REGION Network 2: Block description — Sections 3.2 to 3.7
   // ▂▂▂▂▂▂▂▂▂▂▂▂▂▂▂▂▂▂▂▂▂▂▂▂▂▂▂▂▂▂▂▂▂▂▂▂▂▂▂▂▂▂▂▂
   // 3.2     Warnings and alarms
   // 
   // By default, the block generates 4 alarms and warnings (2 warnings and 2 alarms, 4 in total) 
   // as follows:
   // 
   // 
   //  ――――――――――――――――――――――――――――――――――――――――――
   //  ALARM / WARNING     FUNCTION
   //  ――――――――――――――――――――――――――――――――――――――――――
   //  Alarm high       Scaled signal is equal to or above a preset alarm high setpoint
   //  Warning high      Scaled signal is equal to or above a preset warning high setpoint
   //  Warning low     Scaled signal is equal to or below a preset warning low setpoint
   //  Alarm low      Scaled signal is equal to or below a preset alarm low setpoint
   //  ――――――――――――――――――――――――――――――――――――――――――
   //  Default alarm and warning signals
   // 
   // 
   // The active state of any alarm or warning is stored in the DATA_DYNAMIC structure in the following 
   // variables:
   // 
   //  UT22001_Dy_InstAnalogRead
   //  ――――――――――――――――――――――――――――――――――――――――――
   //  SIGNAL NAME          FUNCTION                     TYPE
   //  ――――――――――――――――――――――――――――――――――――――――――
   //  msg_Alm_H         MESSAGE — Alarm - high alarm is active        Bool
   //  msg_Alm_L          MESSAGE — Alarm - low alarm is active          Bool
   //  msg_Wrn_H          MESSAGE — Warning - high warning is active      Bool
   //  msg_Wrn_L          MESSAGE — Warning - low warning is active        Bool
   //  ――――――――――――――――――――――――――――――――――――――――――
   // 
   // The alarms and warnings that end with _H are activated when the scaled instrument reading is 
   // greater than or equal to a setpoint threshold (i.e. activate when the measured quantity is too 
   // high; generally, if there is both an alarm high and a warning high, the convention within the PAL 
   // is that the warning should activate before the alarm².
   // 
   // 
   // The alarms and warnings that end with _L are activated when the scaled instrument reading is 
   // less than or equal to a setpoint threshold (i.e. activate when the measured quantity is too high; 
   // generally, if there is both an alarm low and a warning low, the convention within the PAL is that 
   // the warning should activate before the alarm².
   // 
   // ――――――――――
   // ²         This is just a convention, there is nothing to stop the warning being set to occur after 
   //      the alarm (i.e. the warning detecting the most extreme condition). All alarms and 
   //      warnings are entirely independent of each other and no error checking is carried 
   //      out to ensure that any particular threshold is above or below another.
   // ――――――――――
   // 
   // All alarms and warnings are individually enabled (a disabled alarm or warning will never be 
   // activated), all alarms and warnings have individual setpoint values (the value at which the 
   // alarm or warning is triggered), all alarms and warnings have individual hysteresis valves 
   // (effectively a tolerance band, the difference between where an alarm activates and where is 
   // deactivates, used to prevent nuisance or “chattering” alarms). Finally, each alarm and warning 
   // has a configurable on and off delay (the alarm or warning will only activate if the reading is 
   // outside the threshold for the on-delay time and similarly will only deactivate when the reading 
   // is inside the threshold and hysteresis for the off-delay time).
   // 
   // The following table summarises all the available signals for each alarm and warning:
   // 
   //  ――――――――――――――――――――――――――――――――――――――――――
   //  SIGNAL          FUNCTION             TYPE   DETAILS
   //  ――――――――――――――――――――――――――――――――――――――――――
   //  CONFIG_XXX_Y_ENABLE Alarm/warning enabled      Bool    1 = enabled, 0 = disabled
   //  SP_XXX_Y_VAL      Alarm/warning setpoint value    Real Engineering units
   //  SP_XXX_Y_HYST_VAL    Alarm/warning hysteresis value Real Engineering units
   //  TIME_XXX_Y_ON_DEL   Alarm/warning on delay time   Real In seconds
   //  TIME_XXX_Y_OFF_DEL     Alarm/warning off delay time   Real In seconds
   //  mode_Xxx_Y_MaskOn     Alarm/warning is masked      Bool    1 = masked, 0 = normal
   //  msg_Xxx_Y         Alarm/warning is active      Bool    1 = active, 0 = inactive
   //  ――――――――――――――――――――――――――――――――――――――――――
   //  Default alarm and warning signals — where XXX is either ALM or WRN and Y is either H or L
   // 
   // 
   // 
   // ▁▁▁▁▁▁▁▁▁▁▁▁▁▁▁▁▁▁▁▁▁▁▁▁▁▁▁▁▁▁▁▁▁▁▁▁▁▁▁▁▁▁▁▁
   // 3.2.1     High alarms and warnings (an example)
   // 
   // This example explains how a high alarm signal is generated, a high warning works in exactly the 
   // same way with WRN being substituted for ALM.
   // 
   // The full set of signals associated with the high alarm are:
   // 
   //  ――――――――――――――――――――――――――――――――――――――――――
   //  SIGNAL           FUNCTION            TYPE   DETAILS
   //  ――――――――――――――――――――――――――――――――――――――――――
   //  SP_ALM_H_VAL      Alarm high setpoint value    Real Engineering units
   //  SP_ALM_H_HYST_VAL    Alarm high hysteresis value Real Engineering units
   //  TIME_ALM_H_ON_DEL   Alarm high on delay time   Real In seconds
   //  TIME_ALM_H_OFF_DEL     Alarm high off delay time   Real In seconds
   //  mode_Alm_H_MaskOn    Alarm is masked         Bool    1 = masked, 0 = normal
   //  msg_Alm_H        Alarm high is active      Bool    1 = active, 0 = inactive
   //  ――――――――――――――――――――――――――――――――――――――――――
   // 
   // The figure below indicates how each of these signal functions (note TIME_ALM_H_ON_DEL and
   // TIME_ALM_H_OFF_DEL have been abbreviated to ON_DEL and OFF_DEL respectively):
   // 
   // 
   //                 │
   //                 │          ╱╲╱╲
   //                 │    ①      ②╱    ╲
   //       SP_ALM_H_VAL↘│____╱╲________╱____________╲③_______④__________ 
   //    SP_ALM_H_HYST_VAL ↕│__╱____╲____╱╎_____╎_______╲____╱╲___________
   //                 │╱    ╲╱ ╎    ╎      ╲╱     ╲
   //                 │        ╎    ╎          ╎╲
   //                 │        ╎    ╎          ╎ ╲___
   //                 │        ╎    ╎          ╎    ╎╲╱
   //                 │    ON_DEL→╎    ╎←    OFF_DEL→╎    ╎←
   //                 ┼─────────────────────────────
   // 
   //                            ╎                        ╎
   // 
   //         msg_Alm_H │             ┏━━━━━━━━━━━━┓
   //                 │             ┃               ┃
   // CONFIG_ALM_H_ENABLE = 1  │             ┃   ALARM IS ACTIVE    ┃
   // & mode_Alm_H_MaskOn = 0 │             ┃               ┃
   //                 │             ┃               ┃
   //                 ┼━━━━━━━━━━━━╶╶╶╶╶╶╶╶╶╶╶╶╶━━━━
   // 
   //                            ╎                        ╎
   // 
   //         msg_Alm_H │          
   // ⑤               │             ╎               ╎             
   // CONFIG_ALM_H_ENABLE = 0  │             
   //     OR          │             ╎               ╎
   // CONFIG_ALM_H_ENABLE = 1  │          
   // & mode_Alm_H_MaskOn = 1 ┼━━━━━━━━━━━━━━━━━━━━━━━━━━━━━
   // 
   // 
   // 
   // ▁▁▁▁▁▁▁▁▁▁▁▁▁▁▁▁▁▁▁▁▁▁▁▁▁▁▁▁▁▁▁▁▁▁▁▁▁▁▁▁▁▁▁▁
   // Scenario ①, alarm setpoint reached, but for less than on-delay duration
   // 
   // The graph represents the scaled analogue instrument reading, actual_Value (in engineering 
   // units). The top horizontal line is the setpoint for the high alarm (SP_ALM_H_VAL).
   // 
   // If the alarm is enabled (CONFIG_ALM_H_ENABLE = 1) then the following actions occur:
   // 
   // At point ① on the graph, the signal actual_Value reaches (and exceeds) the threshold value 
   // SP_ALM_H_VAL; i.e.:
   // 
   //           actual_Value ≥ SP_ALM_H_VAL
   // 
   // At this point, the alarm setpoint is exceeded and the on-delay timer starts; in the case of point ①, 
   // the signal actual_Value falls back below the setpoint value before the on-delay timer reaches 
   // the time set in TIME_ALM_H_ON_DEL, consequently the alarm does not activate.
   // 
   // 
   // 
   // ▁▁▁▁▁▁▁▁▁▁▁▁▁▁▁▁▁▁▁▁▁▁▁▁▁▁▁▁▁▁▁▁▁▁▁▁▁▁▁▁▁▁▁▁
   // Scenario ②, alarm setpoint reached for more than the on-delay duration
   // 
   // At point ② on the graph, the signal actual_Value again reaches (and exceeds) the setpoint value 
   // SP_ALM_H_VAL.
   // 
   // Again, at this point, the alarm threshold is exceeded and the on-delay timer starts; in the case of 
   // point ②, the signal actual_Value remains at or above the setpoint value for the full duration of 
   // the TIME_ALM_H_ON_DEL and consequently the alarm activates (msg_Alm_H goes to a high 
   // state), this is indicated in the middle msg_Alm_H graph.
   // 
   // 
   // 
   // ▁▁▁▁▁▁▁▁▁▁▁▁▁▁▁▁▁▁▁▁▁▁▁▁▁▁▁▁▁▁▁▁▁▁▁▁▁▁▁▁▁▁▁▁
   // Scenario ③, alarm reset level reached, but for less than the off-delay duration
   // 
   // At point ③, the signal actual_Value falls to the point at which the alarm is no longer active i.e.:
   // 
   //           actual_Value < (SP_ALM_H_VAL − SP_ALM_H_HYST_VAL)
   // 
   // Note:    in this case the inequality is less than (not less than or equal to), this is to prevent 
   //      conflict detecting the threshold and detecting the reset value if SP_ALM_H_HYST_VAL 
   //      is set to zero.
   // 
   // At this point, the signal is below the alarm reset level:
   // 
   //           SP_ALM_H_VAL − SP_ALM_H_HYST_VAL
   // 
   // and the off-delay timer starts; in the case of point 3, the signal actual_Value re-turns above the 
   // reset threshold before the off-delay timer reaches the time set in TIME_ALM_H_OFF_DEL, 
   // consequently, the alarm does not deactivate.
   // 
   // 
   // 
   // ▁▁▁▁▁▁▁▁▁▁▁▁▁▁▁▁▁▁▁▁▁▁▁▁▁▁▁▁▁▁▁▁▁▁▁▁▁▁▁▁▁▁▁▁
   // Scenario ④, alarm reset level reached for more than the off-delay duration
   // 
   // At point ④ on the graph, the signal actual_Value again falls below the alarm reset level 
   // (SP_ALM_H_VAL − SP_ALM_H_HYST_VAL).
   // 
   // Again, at this point, the off-delay timer starts; in the case of point ④, the signal actual_Value 
   // remains below the reset threshold for the full duration of the TIME_ALM_H_OFF_DEL and 
   // consequently, the alarm deactivates (msg_Alm_H goes to a low state), this is indicated in the 
   // middle msg_Alm_H graph.
   // 
   // 
   // 
   // ▁▁▁▁▁▁▁▁▁▁▁▁▁▁▁▁▁▁▁▁▁▁▁▁▁▁▁▁▁▁▁▁▁▁▁▁▁▁▁▁▁▁▁▁
   // Scenario ⑤, alarm is disabled
   // 
   // If the alarm is disabled (CONFIG_ALM_H_ENABLE = 0) then the alarm will never activate 
   // (msg_Alm_H is always in a low state), this is indicated in the lower msg_Alm_H graph.
   // 
   // Note:    The timer for disabled alarms and warnings is permanently set to zero.
   // 
   // 
   // ▁▁▁▁▁▁▁▁▁▁▁▁▁▁▁▁▁▁▁▁▁▁▁▁▁▁▁▁▁▁▁▁▁▁▁▁▁▁▁▁▁▁▁▁
   // 3.2.2     Low alarms and warnings
   // 
   // Low alarms and warnings are very similar to the high alarms of § 3.2.1, they do however work
   // in the opposite sense (the inequalities are reversed), low alarms and warnings are activated
   // when the actual_Value falls below, or is equal to, the SP_ALM_L_VAL, and deactivates when it
   // rises above SP_ALM_L_VAL + SP_ALM_L_HYST_VAL.
   // 
   // On and off delays work in exactly the same way as those for the high alarm.
   // 
   // A worked example of the low alarm is given in the online documentation for this block:
   // 
   // select this block in the project tree and press:
   //      SHIFT + F1
   // 
   // 
   // 
   // 
   // ▁▁▁▁▁▁▁▁▁▁▁▁▁▁▁▁▁▁▁▁▁▁▁▁▁▁▁▁▁▁▁▁▁▁▁▁▁▁▁▁▁▁▁▁
   // 3.2.3     Masking alarms and warnings
   // 
   // There are conditions where it can become necessary to mask (supress) alarms and warnings, a 
   // typical example could be a flow meter that monitors the flow into a filter; under normal 
   // conditions the flow meter would generate a low alarm if the flow into the filter were below a 
   // certain setpoint (indicating that the filter is becoming blocked).
   // 
   // It would be normal practice to supress this alarm when the filter was being cleaned, under 
   // these circumstances there would be no flow into the filter, but this would be a normal operating 
   // condition for the filter; the flow meter should only be monitoring for a low alarm during normal 
   // operation, not when the filter is being cleaned.
   // 
   // This suppression of an alarm or warning is referred to as “masking”, and there is a mask bit for 
   // each alarm and warning:
   // 
   //  ――――――――――――――――――――――――――――――――――――――――――
   //  SIGNAL           FUNCTION           TYPE   DETAILS
   //  ――――――――――――――――――――――――――――――――――――――――――
   //  mode_Alm_H_MaskOn    Masks the high alarm     Bool    1 = alarm masked, 0 = normal
   //  mode_Alm_L_MaskOn    Masks the low alarm    Bool    1 = alarm masked, 0 = normal
   //  mode_Wrn_H_MaskOn    Masks the high warning    Bool    1 = warning masked, 0 = normal
   //  mode_Wrn_L_MaskOn     Masks the low warning      Bool    1 = warning masked, 0 = normal
   //  ――――――――――――――――――――――――――――――――――――――――――
   //  Alarm and warning mask signals
   // 
   //  
   // Any alarm or warning that is masked (the mode_Xxx_Y_MaskOn = 1), will deactivate instantly 
   // (there is no off-delay) and will not reactivate activate (the msg_Xxx_Y will be set to zero), the 
   // effect is the same as if the CONFIG_XXX_Y_ENABLE bit were turned off.
   // 
   // The difference between the mask and the ENABLE signals is that the enable signal is a 
   // configuration of the instrument (it determines which alarms and warnings are configured for the 
   // particular instrument) and does not change at run-time (it is stored in static data block).
   // 
   // The mask signal on the other hand can be changed at run-time (either by some aspect of the 
   // Controller program or by the operator). The mask signal is stored in a dynamic data block and 
   // can be freely modified.
   // 
   // Note:    If an alarm or warning is not enabled (CONFIG_XXX_Y_ENABLE = 0), then the mask bit 
   //      (mode_Xxx_Y_MaskOn) will not do anything (setting it will not enable the alarm), in 
   //      fact if the alarm or warning is not enabled, the mask bit will be permanently set to 
   //      zero.
   // 
   // Masking alarms and warnings is the correct way to disable an alarm as part of the process 
   // operation of the plant.
   // 
   // When an alarm or warning goes from a masked condition to an unmasked condition (returns to 
   // normal operation), the on-delay timer will be reset and any alarm or warning condition will 
   // have to go back through the on-delay process before the alarm or warning can reactivate, this is 
   // true even if the alarm were active before being masked.
   // 
   // 
   // 
   // 
   // ▁▁▁▁▁▁▁▁▁▁▁▁▁▁▁▁▁▁▁▁▁▁▁▁▁▁▁▁▁▁▁▁▁▁▁▁▁▁▁▁▁▁▁▁
   // 3.2.4     A note on dynamically enabling alarms
   // 
   // In normal operations, alarms are either enabled or disabled as part of the instrument 
   // configuration and this configuration will not change during run-time; the enable signal 
   // (CONFIG_XXX_Y_ENABLE) is after all in a static data block. 
   // 
   // However, it is possible that the static data block is being used as a recipe block and as such it 
   // could be overloaded at some point during run-time.
   // 
   // Should the block detect a change in any of the CONFIG_XXX_Y_ENABLE; specifically, a rising 
   // edge, the block provided error checking to ensure that the associated alarm/warning timer 
   // (actual_Xxx_Y_Timer) is preset to correct TIME_XXX_Y_ON_DEL, this prevents the alarm/warning 
   // from activating instantly, if the actual_Value is outside the alarm/warning setpoint. A condition 
   // that could arise because the timer is set to zero while ever the alarm/warning is disabled.
   // 
   // Note:    This is a minor technical point, but it is a necessary error trapping mechanism — the 
   //      situation could arise even if it is unlikely.
   // 
   // 
   // 
   // ▂▂▂▂▂▂▂▂▂▂▂▂▂▂▂▂▂▂▂▂▂▂▂▂▂▂▂▂▂▂▂▂▂▂▂▂▂▂▂▂▂▂▂▂
   // 3.3     Fault signals
   // 
   // There are four fault signals that can be produced by the block:
   // 
   // 
   //  ――――――――――――――――――――――――――――――――――――――――――
   //  SIGNAL           FUNCTION            TYPE   DETAILS
   //  ――――――――――――――――――――――――――――――――――――――――――
   //  msg_Flt_UnderRange   The instrument is more than   Bool    1 = under range, 0 = healthy
   //                 a percentage below the its 
   //                 minimum value
   //  msg_Flt_OverRange     The instrument is more than   Bool    1 = over range, 0 = healthy
   //                 a percentage above its 
   //                 maximum value
   //  msg_Flt_OutOfRange   Common fault, either       Bool    1 = out of range, 0 = healthy
   //                 under or over range
   //  msg_Flt_External     The instrument itself is    Bool    1 = fault, 0 = healthy
   //                 indicating a fault 
   //                 (hardwired signal)
   //  ――――――――――――――――――――――――――――――――――――――――――
   //  Block fault signals 
   // 
   // 
   // 
   // ▁▁▁▁▁▁▁▁▁▁▁▁▁▁▁▁▁▁▁▁▁▁▁▁▁▁▁▁▁▁▁▁▁▁▁▁▁▁▁▁▁▁▁▁
   // 3.3.1     Over, under and out of range fault signals
   // 
   // If the signal from the instrument the RAW_ANALOG signal, is outside the RANGE_RAW_MIN to 
   // RANGE_RAW_MAX range (red dotted area of the graph, Figure 3.1), the scaled instrument reading 
   // (actual_Value) will still be calculated correctly; however, an appropriate, over-range or 
   // under-range (msg_Flt_OverRange or msg_Flt_UnderRange) signal will be generated to indicate 
   // that the instrument signal is outside of its calibrated range and is potentially no longer accurate.
   // 
   // Some tolerance is permitted before either the msg_Flt_OverRange or msg_Flt_UnderRange 
   // signals is activated (this is to prevent nuisance alarms — most instruments are tolerant of slight 
   // over and under shoot readings). 
   // 
   // The tolerance applied to the out of range signals is a percentage of the raw range of the 
   // instrument (the raw range being RANGE_RAW_MAX − RANGE_RAW_MIN). 
   // 
   // The tolerance to be applied is given in the parameter RANGE_OOR_PERCENT, this is a real 
   // (floating point) number in the range 0.0-10.0%.
   // 
   // If the tolerance for the instrument is not known, a generic value of 2.5% should be used.
   // 
   // The out of range tolerance absolute value (in terms of the RAW_ANALOG rather than as a 
   // percentage) is calculated as:
   // 
   // 
   // 
   // ┌─────────────────────────────────────┐
   // │                            (RANGE_RAW_MAX ─ RANGE_RAW_MIN) ╳ RANGE_OOR_PERCENT  │
   // │ calcRawOOR =  ―――――――――――――――――――――――――――― │
   // │                      100              │
   // └─────────────────────────────────────┘
   // 
   // Thus, if RANGE_RAW_MIN is 0, RANGE_RAW_MAX is 27648 and a RANGE_OOR_PERCENT of 2.5% is 
   // selected, the absolute out of range value (calcRawOOR in the above equation) has a calculated
   //  value of 691. 
   // 
   // In this example, the msg_Flt_OverRange signal would activate when RAW_ANALOG 
   // exceeded a value of RANGE_RAW_MAX + 691 (or 28,339). The msg_Flt_UnderRange signal would 
   // activate when RAW_ANALOG fell below a value of RANGE_RAW_MIN − 691 (or −691).
   // 
   // The RANGE_OOR_PERCENT is applied directly to the RAW_ANALOG signal, however, because the 
   // instrument is considered to be linear, the same calculation can also be ap-plied directly to the 
   // scaled reading of the instrument (actual_Value). 
   // 
   // In the example given in § 2.1, the instrument spans the range of -100 l/s to +100 l/s 
   // (i.e. RANGE_SCALE_MIN = -100 and RANGE_SCALE_MAX = +100) then the scaled range of the 
   // instrument is 200 l/s (RANGE_SCALE_MAX − RANGE_SCALE_MIN) and the absolute out of range 
   // value would be 2.5% of the scaled range (or 5 l/s). thus, the msg_Flt_OverRange signal would 
   // activate above 105 l/s and the msg_Flt_UnderRange signal would activate below −105 l/s.
   // 
   // Note:    If the range information supplied to the module is incorrect, either:
   //        •   RAW_MAX <= RAW_MIN or
   //        •   SCALE_MAX <= SCALE_MIN
   //      Then all the out of range signals are activated
   // 
   // 
   // 
   // ▁▁▁▁▁▁▁▁▁▁▁▁▁▁▁▁▁▁▁▁▁▁▁▁▁▁▁▁▁▁▁▁▁▁▁▁▁▁▁▁▁▁▁▁
   // Common out of range signal
   // 
   // There is a third out of range signal: msg_Flt_OutOfRange, this signal is a common signal that 
   // just indicates the instrument is out of its calibrated range (it does not specify whether it is over 
   // or under range). It is activated if either the msg_Flt_OverRange or msg_Flt_UnderRange signal is 
   // active.
   // 
   // 
   // 
   // ▁▁▁▁▁▁▁▁▁▁▁▁▁▁▁▁▁▁▁▁▁▁▁▁▁▁▁▁▁▁▁▁▁▁▁▁▁▁▁▁▁▁▁▁
   // 3.3.2     External fault signal
   // 
   // The external fault is an optional hardwired signal from the instrument, it indicates that the 
   // instrument itself is registering that there is some problem. Such external fault signals are more 
   // commonly associated with complex instruments (mass flow metres, ultrasonic level 
   // transducers, analytical instruments &c.) rather than the more simplistic instruments (pressure 
   // sensors, temperature transmitters &c.).
   // 
   // Typical examples of external faults would be:
   // 
   //    •   No medium present in a mass flow meter (if the instrument were measuring liquid 
   //      flow and the pipe had become empty)
   // 
   //    •   Foam indication from an ultrasonic level transducer (preventing an accurate level 
   //      reading)
   // 
   // Such fault signals are generally indicated via a hardwired digital input to the Controller.
   // 
   // The external fault signal (if used) is passed to the block as the parameter: EXT_FAULT
   // 
   //  ――――――――――――――――――――――――――――――――――――――――――
   //  PARAMETER          FUNCTION            TYPE   DETAILS
   //  ――――――――――――――――――――――――――――――――――――――――――
   //  EXT_FAULT        Hardwired signal indicating    Bool    1 = fault, 0 = healthy
   //                 the instrument is in a fault 
   //                 condition
   //  ――――――――――――――――――――――――――――――――――――――――――
   //  Block external fault parameter 
   // 
   // If the EXT_FAULT signal is not required, the input should be set to _false.
   // 
   // If the instrument generates a fault signal in the opposite sense, i.e. 0 = fault and 1 = healthy (this 
   // is a common fail-safe condition, that generates a fault signal if the instrument is disconnected 
   // or a wire break occurs), then a normally closed contact should be applied to the EXT_FAULT 
   // parameter to invert the signal into the block (see Figure 3.4):
   // 
   // 
   //                       ┌─────────────
   //    ───────────────────┤ FC02001 
   //                       ├───────────────┤
   //                           "FC001" ─┤ RAW_ANALOG           │
   //                       │               │
   //         "FC001_FAULT"           │               │
   //      ────┤╱├──────────┤ EXT_FAULT                │
   //                       │               │
   //                       │               │
   //   "DB02001_St_StdInstAnalogRead".FC001 ─┤ STATIC_DATA             │
   //                       │
   //   "DB22001_Dy_StdInstAnalogRead".FC001 ─┤ DYNAMIC_DATA
   //                       │
   //                       │
   // 
   // 
   // If the EXT_FAULT parameter is activated (set to 1), the corresponding fault signal within the 
   // dynamic data (msg_Flt_External) will be activated, there are no delays or other filtering 
   // associated with this signal.
   // 
   // Note:    The external fault does not in any way impact the reading and scaling of the 
   //      instrument or the production of any alarms or warnings.
   // 
   // 
   // 
   // ▂▂▂▂▂▂▂▂▂▂▂▂▂▂▂▂▂▂▂▂▂▂▂▂▂▂▂▂▂▂▂▂▂▂▂▂▂▂▂▂▂▂▂▂
   // 3.4     Operating mode
   // 
   // This block  supports various operating modes:
   // 
   //    •   Simulation mode
   //    •   Remote/local mode
   //    •   Faceplate disabled mode
   // 
   // Examining these in turn:
   // 
   // 
   // ▁▁▁▁▁▁▁▁▁▁▁▁▁▁▁▁▁▁▁▁▁▁▁▁▁▁▁▁▁▁▁▁▁▁▁▁▁▁▁▁▁▁▁▁
   // 3.4.1     Simulation mode
   // 
   // The instrument can be switched to a simulation mode, in which the actual reading from the 
   // instrument is replaced by a simulated value provided by the operator. 
   // 
   // Simulation mode is generally used during testing, but can also be applied in a process 
   // environment if a fault condition is detected within the instrument; this scenario allows the plant 
   // to continue operating (albeit under some degree of manual control) until the instrument is 
   // repaired or replaced.
   // 
   // The following data points are associated with the simulation mode:
   // 
   //  ――――――――――――――――――――――――――――――――――――――――――
   //  SIGNAL           FUNCTION            TYPE   DETAILS
   //  ――――――――――――――――――――――――――――――――――――――――――
   //  CONFIG_SIM_DISABLE      Prevents simulation mode   Bool    1 = no sim, 0 = sim permitted
   //                 being activated under all 
   //                 circumstances
   // 
   //  mode_SimOn        Activates simulation mode,    Bool    1 = sim on, 0 = sim off
   //                 if active, the scaled reading 
   //                 of the instrument (Value) will 
   //                 be set to mode_SimValue
   // 
   //  mode_SimValue      Scaled instrument reading   Real    Simulated instrument value
   //                 (Value) will be set to this if 
   //                 simulation mode is on
   //                 (CONFIG_SIM_OFF = 0 and 
   //                 mode_SimOn = 1)
   // 
   //  status_SimOn       Status indication, shows if    Bool    1 = sim active, 0 = Sim off
   //                 simulation mode is active
   //  ――――――――――――――――――――――――――――――――――――――――――
   // 
   // 
   // Simulation mode can only be activated by the operator via a faceplate available at the 
   // supervisory system (SCADA/HMI).
   // 
   // If simulation mode is disabled (configuration signal CONFIG_SIM_OFF is set to 1), then the 
   // simulation mode cannot be turned on under any circumstances, the option is greyed out on the 
   // supervisory system faceplate and the block will constantly reset the mode_SimOn signal.
   // 
   // If simulation mode is permitted (CONFIG_SIM_OFF = 0), then setting mode_SimOn to 1 will 
   // activate simulation mode and the scaled instrument value (actual_Value) will be set to the 
   // value stored in mode_SimValue:
   // 
   //           i.e. actual_Value = mode_SimValue
   // 
   // and all fault messages will be reset.
   // 
   // The operator can set and adjust the simulation value (mode_SimValue) from the instrument
   // faceplate on the supervisory system. The simulation value can be adjusted at any time by the 
   // operator (even if simulation mode has not been activated), but will not be applied until 
   // simulation mode is turned on (mode_SimOn = 1). 
   // 
   // If simulation mode is completely disabled (CONFIG_SIM_OFF is set to 1) then the operator will
   // not be able to adjust the simulated value (mode_SimValue will be greyed out on the faceplate).
   // 
   // 
   // 
   // ▁▁▁▁▁▁▁▁▁▁▁▁▁▁▁▁▁▁▁▁▁▁▁▁▁▁▁▁▁▁▁▁▁▁▁▁▁▁▁▁▁▁▁▁
   // 3.4.2     Remote/local mode
   // 
   // Remote and local operating modes refer to the supervisory system that has control of the 
   // instrument (i.e. which system can write to the device and change the operating mode of the 
   // device). 
   // 
   // This type of mode is usual present where a plant has a remote central control location (a control 
   // room) that normally controls the device (remote control), but also has a field panel with a local 
   // HMI that an operator in the field can select to take over control of the device (local control) for 
   // maintenance purposes.
   // 
   // The modes are as follows (and are mutually exclusive, only one will be active):
   // 
   //    Remote        Only the remote system in the control room can 
   //                 control the device
   // 
   //    Local            A local system has taken control of the device and the remote 
   //                 system can no longer issue commands to it
   // 
   //    Remote/local disabled   The system does not use remote/local modes and any 
   //      (ALL mode)     supervisory system can issue commands to the device 
   //  
   // Remote/local control is generally handled by the supervisory systems themselves; however, the 
   // supervisory systems need a storage area per device to record which mode that device is in, local 
   // control is often activated by a panel key-switch, that changes the state of several devices from 
   // remote to local (usually all the devices controlled by the local panel).
   // 
   // The block simply identifies the remote/local mode from the mode signals and configuration 
   // signals provided to the block.
   // 
   // For systems that do not use remote/local modes (any supervisory system can control the device, 
   // or control is determined by operator privileges), the remote/local modes can be disabled 
   // (CONFIG_RL_ENABLE is set to zero) and the device is effectively in ALL mode (any system can 
   // control the device).
   // 
   // If remote/local operation is in use, the supervisory system that does not have control will still 
   // display all the information from the device, but will not be able to control the device (it could not 
   // for example, activate simulation mode) and all control function (faceplate functions) will be 
   // greyed out.
   // 
   // The following signals are associated with remote/local/all modes:
   // 
   // 
   //  ――――――――――――――――――――――――――――――――――――――――――
   //  SIGNAL           FUNCTION            TYPE   DETAILS
   //  ――――――――――――――――――――――――――――――――――――――――――
   //  CONFIG_RL_ENABLE   Allows Remote and Local      Bool    1 = Remote/local selected
   //                 modes to be selected        0 = All mode is active
   // 
   //  mode_RemoteOn       Activates remote mode     Bool    1 = remote mode on, 
   //                 CONFIG_RL_ENABLE must = 1    0 = remote mode off
   // 
   //  mode_LocalOn     Activates local mode          Bool    1 = local mode on, 
   //                 CONFIG_RL_ENABLE must = 1    0 = remote mode off
   // 
   //  status_RemoteOn      Status remote mode on     Bool    1 = remote mode on, 
   //                               0 = remote mode off
   // 
   //  status_LocalOn       Status local mode on      Bool 1 = local mode on, 
   //                               0 = local mode off
   // 
   //  status_RLOff       Status ALL mode is on = 0    Bool 1 = ALL mode on, 
   //                               0 = ALL mode off
   //  ――――――――――――――――――――――――――――――――――――――――――
   //  Block remote/local signals 
   // 
   // By default, remote/local is disabled — ALL mode is selected (CONFIG_RL_ENABLE = 0).
   // 
   // 
   // 
   // 
   // ▁▁▁▁▁▁▁▁▁▁▁▁▁▁▁▁▁▁▁▁▁▁▁▁▁▁▁▁▁▁▁▁▁▁▁▁▁▁▁▁▁▁▁▁
   // 3.4.3     Faceplate disable mode
   // 
   // It is possible to disable the supervisory system faceplate from within the block, the con-figuration 
   // signal:
   // 
   // 
   //  ――――――――――――――――――――――――――――――――――――――――――
   //  SIGNAL           FUNCTION            TYPE   DETAILS
   //  ――――――――――――――――――――――――――――――――――――――――――
   //  CONFIG_FP_DISABLE     Disable the supervisory      Bool    1 = Faceplate disabled
   //                 system faceplate           0 = normal
   //  ――――――――――――――――――――――――――――――――――――――――――
   //  Block faceplate disable signal 
   // 
   // If the faceplate is disabled (CONFIG_FP_DISABLE = 1), the supervisory system will not allow the 
   // device faceplate to be opened (normally achieved by clicking the block icon or device symbol), 
   // this in turn prevents the operator from affecting the device in anyway, it would not, for example, 
   // be possible to put the device into simulation mode.
   // 
   // Similarly, if the faceplate is disabled, the module will set remote/local mode to ALL and will 
   // disable simulation mode.
   // 
   // 
   // 
   // ▂▂▂▂▂▂▂▂▂▂▂▂▂▂▂▂▂▂▂▂▂▂▂▂▂▂▂▂▂▂▂▂▂▂▂▂▂▂▂▂▂▂▂▂
   // 3.5     Block icon signals
   // 
   // This block has a partner block icon that represents the instrument and its various modes and 
   // status in a graphical format (block icon) that is displayed on a supervisory system (SCADA or HMI).
   // 
   // See the online documentation for this block — select the block in the project tree and press:
   //      SHIFT + F1
   // 
   // The supervisory system interface is available in section 3.7 of the online SMDS document.
   // 
   // 
   // 
   // ▁▁▁▁▁▁▁▁▁▁▁▁▁▁▁▁▁▁▁▁▁▁▁▁▁▁▁▁▁▁▁▁▁▁▁▁▁▁▁▁▁▁▁▁
   // 3.5.1     Understanding status signals
   // 
   // The status signals for faults, alarms and warnings are either duplicates of the message signals 
   // (signals beginning with msg_) or logical combinations of them.
   // 
   // The following is a full list of the status signals:
   // 
   //  ――――――――――――――――――――――――――――――――――――――――――
   //  SIGNAL           FUNCTION            TYPE   DETAILS
   //  ――――――――――――――――――――――――――――――――――――――――――
   //  status_Alm_H        Identical to: msg_Alm_H    Bool    1 = high alm active, 0 = no alm
   // 
   //  status_Alm_L         Identical to: msg_Alm_L       Bool    1 = low alm active, 0 = no alm
   // 
   //  status_Wrn_H        Identical to: msg_Wrn_H    Bool    1 = high wrn active, 0 = no wrn
   // 
   //  status_Wrn_L         Identical to: msg_Wrn_L     Bool    1 = low wrn active, 0 = no wrn
   // 
   //  status_Alm_H_Mask     High alarm is masked     Bool    1 = masked, 0 = normal
   // 
   //  status_Alm_L_Mask   Low alarm is masked      Bool    1 = masked, 0 = normal
   // 
   //  status_Wrn_H_Mask      High warning is masked    Bool    1 = masked, 0 = normal
   // 
   //  status_Wrn_L_Mask       Low warning is masked     Bool    1 = masked, 0 = normal
   // 
   //  status_Alm_H_Dis         High alarm is disabled       Bool    1 = disabled, 0 = normal
   // 
   //  status_Alm_L_Dis       Low alarm is disabled        Bool    1 = disabled, 0 = normal
   // 
   //  status_Wrn_H_Dis          High warning is disabled      Bool    1 = disabled, 0 = normal
   // 
   //  status_Wrn_L_Dis           Low warning is disabled       Bool    1 = disabled, 0 = normal
   // 
   //  status_Fault       Indicates any of the msg_Flt    Bool    1 = fault active, 0 = healthy
   //                 signals are active:
   //                  msg_Flt_UnderRange
   //                  msg_Flt_OverRange
   //                  msg_Flt_OutOfRange
   //                  msg_Flt_External 
   // 
   //  status_SimOn       Status simulation mode on     Bool    1 = sim on, 0 = sim off
   // 
   //  status_RemoteOn      Status remote mode on     Bool    1 = rem on, 0 = rem off
   // 
   //  status_LocalOn       Status local mode on      Bool    1 = loc on, 0 = loc off 
   // 
   //  status_RLOff       Status ALL mode is on           Bool    1 = ALL mode on, 
   //                               0 = ALL mode off
   //  ――――――――――――――――――――――――――――――――――――――――――
   //  Block status signals 
   // 
   // 
   // 
   // ▁▁▁▁▁▁▁▁▁▁▁▁▁▁▁▁▁▁▁▁▁▁▁▁▁▁▁▁▁▁▁▁▁▁▁▁▁▁▁▁▁▁▁▁
   // 3.5.2     String constants for tag name and units
   // 
   // The STATIC_DATA structure holds two string values:
   // 
   //  UT02001_St_InstAnalogRead (full contents)
   //  ――――――――――――――――――――――――――――――――――――――――――
   //  SIGNAL NAME          FUNCTION                     TYPE
   //  ――――――――――――――――――――――――――――――――――――――――――
   //  INFO_TAG          INFORMATION — Instrument ID tag          String[20]
   // 
   //  INFO_UNITS          INFORMATION — Engineering units of the instrument  String[10]
   //                        (unit of measure)
   //  ――――――――――――――――――――――――――――――――――――――――――
   //  String constants for the instrument
   // 
   // These two strings allow the supervisory system to populate the instrument tag (e.g. FIC001) and 
   // the engineering units applicable to the instrument (L/s for example) directly from the data 
   // stored in the PLC; it means the block icon can be used directly within the supervisory system 
   // graphic without customisation; all the data will be populated directly at runtime.
   // 
   //                ━━━   ⬙⬙⬙⬙⬙⬙   ━━━
END_REGION

REGION Network 3: Block description — Sections 4 to 11
   // ▄▄▄▄▄▄▄▄▄▄▄▄▄▄▄▄▄▄▄▄▄▄▄▄▄▄▄▄▄▄▄▄▄▄▄▄▄▄▄▄▄▄▄▄
   // 4.     PARAMETERS
   // 
   // 
   // The following parameters are associated with the block:
   // 
   //  
   //  ――――――――――――――――――――――――――――――――――――――――――
   //  PARAM         FUNCTION                    TYPE      IN-OUT 
   //  ――――――――――――――――――――――――――――――――――――――――――
   //  SYS_SIGNALS      Common system signals              UT21000    In
   //           logic and timing signals for parametric access
   // 
   //  RAW_ANALOG      The unscaled analogue input (input word         Word     In
   //           address for the IO card to which the instrument 
   //           is connected)
   // 
   //  EXT_FAULT     Optional external fault signal for the instrument      Bool      In
   //           (1 = fault, 0 = healthy). If not required, set 
   //           permanently to _False
   // 
   //  STATIC_DATA     Data structure that holds the configuration data     UT02001    In
   //           for the instrument (raw range, scaled range 
   //           alarm and warning values, filtering times, 
   //           hysteresis values &c.)
   // 
   //  DYNAMIC_DATA      Data structure that holds the live data for the       UT22001    InOut
   //           instrument (its reading in engineering units, 
   //           any alarms or warnings that may be active, 
   //           current timer values, selected operating 
   //           mode &c.)
   //  ――――――――――――――――――――――――――――――――――――――――――
   // 
   //                ━━━   ⬙⬙⬙⬙⬙⬙   ━━━
   // 
   // 
   // 
   // ▄▄▄▄▄▄▄▄▄▄▄▄▄▄▄▄▄▄▄▄▄▄▄▄▄▄▄▄▄▄▄▄▄▄▄▄▄▄▄▄▄▄▄▄
   // 5.     DATA STRUCTURES AND USAGE (AND INSTANCE DATA BLOCKS)
   // 
   // 
   // The block has the following associated data structure:
   // 
   // 
   //  ――――――――――――――――――――――――――――――――――――――――――
   //  DATA STRUCTURE             DESCRIPTION
   //  ――――――――――――――――――――――――――――――――――――――――――
   //  UT01000_St_SysRevision          Revision information for this block    See FC01001
   //  UT01001_St_SysLicence           Licence information for this block  See FC01001
   //  UT21000_Dy_SysSignals           System signals for logic and timing  See FC01001
   // 
   //  UT02001_St_InstAnalogRead      Static data structure for an analogue instrument.
   //                     Holds configuration information, instrument ranges 
   //                     and scaling, alarm/warning thresholds &c.
   // 
   //  UT22001_Dy_InstAnalogRead        Dynamic data structure for an analogue instrument.
   //                     Current scaled instrument reading, alarm status, 
   //                     operating modes, timer values &c.
   //  ――――――――――――――――――――――――――――――――――――――――――
   // 
   // 
   // 
   // ▂▂▂▂▂▂▂▂▂▂▂▂▂▂▂▂▂▂▂▂▂▂▂▂▂▂▂▂▂▂▂▂▂▂▂▂▂▂▂▂▂▂▂▂
   // 5.1     UT02001_St_InstAnalogRead
   // 
   // The static data structure for an analogue instrument.
   // 
   // 
   //  UT02001_St_InstAnalogRead (full contents)
   //  ――――――――――――――――――――――――――――――――――――――――――
   //  SIGNAL NAME          FUNCTION                     TYPE
   //  ――――――――――――――――――――――――――――――――――――――――――
   //  CONFIG_ALM_H_ENABLE  CONFIG — High alarm is enabled          Bool
   //                      (1 = enabled, 0 = no alarm) 
   //  CONFIG_ALM_L_ENABLE   CONFIG — Low alarm is enabled           Bool
   //                      (1 = enabled, 0 = no alarm)
   //  CONFIG_WRN_H_ENABLE     CONFIG — High warning is enabled         Bool
   //                      (1 = enabled, 0 = no warning)
   //  CONFIG_WRN_L_ENABLE     CONFIG — Low warning is enabled          Bool
   //                      (1 = enabled, 0 = no warning)
   //  CONFIG_FP_DISABLE      CONFIG — Faceplate is disabled           Bool
   //                      (1 = no Faceplate, 0 = normal)
   //  CONFIG_SIM_DISABLE    CONFIG — Simulation is disabled            Bool
   //                      (1 = no Simulation, 0 = normal)
   //  CONFIG_RL_ENABLE    CONFIG — Remote/local mode enabled       Bool
   //                      (1 = enabled, 0 = all mode)
   // 
   //  RANGE_RAW_MIN       RANGE — Minimum value of the raw analogue    Int
   //                     signal (at the card)
   //  RANGE_RAW_MAX      RANGE — Maximum value of the raw analogue      Int
   //                     signal (at the card)
   //  RANGE_SCALE_MIN      RANGE — Minimum value of the scaled analogue     Real
   //                     signal [engineering units]
   //  RANGE_SCALE_MAX     RANGE — Maximum value of the scaled analogue    Real
   //                     signal [engineering units]
   //  RANGE_OOR_PERCENT      RANGE — Out of range percentage, beyond which    Real
   //                     the instrument is out of range
   // 
   //  INFO_TAG          INFORMATION — Instrument ID tag          String[20]
   // 
   //  INFO_UNITS          INFORMATION — Engineering units of the instrument  String[10]
   //                        (unit of measure)
   // 
   //  SP_ALM_H_VAL       SETPOINT — High alarm threshold value         Real
   //                      [engineering units]
   //  SP_ALM_L_VAL       SETPOINT — Low alarm threshold value       Real
   //                      [engineering units]
   //  SP_WRN_H_VAL         SETPOINT — High warning threshold value        Real
   //                      [engineering units]
   //  SP_WRN_L_VAL       SETPOINT — Low warning threshold value      Real
   //                      [engineering units]
   //  SP_ALM_H_HYST_VAL     SETPOINT — High alarm hysteresis value        Real
   //                      [engineering units]
   //  SP_ALM_L_HYST_VAL     SETPOINT — Low alarm hysteresis value         Real
   //                      [engineering units]
   //  SP_WRN_H_HYST_VAL    SETPOINT — High warning hysteresis value       Real
   //                      [engineering units]
   //  SP_WRN_L_HYST_VAL     SETPOINT — Low warning hysteresis value        Real
   //                      [engineering units]
   // 
   //  TIME_ALM_H_ON_DEL    TIMER — High alarm on delay time          Real
   //                      (activation delay), [seconds]
   //  TIME_ALM_L_ON_DEL     TIMER — Low alarm on delay time           Real
   //                      (activation delay), [seconds]
   //  TIME_WRN_H_ON_DEL       TIMER — High warning on delay time         Real
   //                      (activation delay), [seconds]
   //  TIME_WRN_L_ON_DEL        TIMER — Low warning on delay time          Real
   //                      (activation delay), [seconds]
   //  TIME_ALM_H_OFF_DEL      TIMER — High alarm off delay time           Real
   //                      (deactivation delay), [seconds]
   //  TIME_ALM_L_OFF_DEL       TIMER — Low alarm off delay time            Real
   //                      (deactivation delay), [seconds]
   //  TIME_WRN_H_OFF_DEL      TIMER — High warning off delay time          Real
   //                      (deactivation delay), [seconds]
   //  TIME_WRN_L_OFF_DEL      TIMER — Low warning off delay time           Real
   //                      (deactivation delay), [seconds]
   //  ――――――――――――――――――――――――――――――――――――――――――
   // 
   // 
   // 
   // ▂▂▂▂▂▂▂▂▂▂▂▂▂▂▂▂▂▂▂▂▂▂▂▂▂▂▂▂▂▂▂▂▂▂▂▂▂▂▂▂▂▂▂▂
   // 5.2      UT22001_Dy_InstAnalogRead
   // 
   // The static data structure for an analogue instrument.
   // 
   // 
   // 
   //  UT22001_Dy_InstAnalogReadl (full contents)
   //  ――――――――――――――――――――――――――――――――――――――――――
   //  SIGNAL NAME          FUNCTION                     TYPE
   //  ――――――――――――――――――――――――――――――――――――――――――
   //  status_ConfigError       STATUS — Raw or scaled range configuration error   Bool
   //                      (1 = Config error, 0 = OK)
   //  status_Alm_H         STATUS — High alarm is active           Bool
   //                      (1 = alarm active, 0 = no alarm)
   //  status_Alm_L          STATUS — Low alarm is active            Bool
   //                      (1 = alarm active, 0 = no alarm)
   //  status_Wrn_H         STATUS — High warning is active          Bool
   //                      (1 = warning active, 0 = no warning)
   //  status_Wrn_L          STATUS — Low warning is active           Bool
   //                      (1 = warning active, 0 = no warning)
   //  status_Alm_H_Mask       STATUS — High alarm is masked             Bool
   //                      (1 = alarm masked, 0 = normal)
   //  status_Alm_L_Mask        STATUS — Low alarm is masked              Bool
   //                      (1 = alarm masked, 0 = normal)
   //  status_Wrn_H_Mask       STATUS — High warning is masked            Bool
   //                      (1 = warning masked, 0 = normal)
   //  status_Wrn_L_Mask        STATUS — Low warning is masked             Bool
   //                      (1 = warning masked, 0 = normal)
   //  status_Alm_H_Dis           STATUS — High alarm is disabled            Bool
   //                      (1 = alarm disabled, 0 = normal)
   //  status_Alm_L_Dis            STATUS — Low alarm is disabled             Bool
   //                      (1 = alarm disabled, 0 = normal)
   //  status_Wrn_H_Dis           STATUS — High warning is disabled           Bool
   //                      (1 = warning disabled, 0 = normal)
   //  status_Wrn_L_Dis            STATUS — Low warning is disabled            Bool
   //                      (1 = warning disabled, 0 = normal)
   //  status_Fault            STATUS — Instrument is in fault             Bool
   //                      (1 = fault present, 0 = healthy)
   //  status_SimOn           STATUS — Instrument is in simulation mode     Bool
   //                      (1 = Simulation mode, 0 = normal)
   //  status_RemoteOn       STATUS — Instrument is in remote mode        Bool
   //                      (1 = Remote mode, 0 = normal)
   //  status_LocalOn         STATUS — Instrument is in local mode          Bool
   //                      (1 = Local mode, 0 = normal)
   //  status_RLOff         STATUS — Instrument is in ALL mode         Bool
   //                      (1 = ALL mode, 0 = normal)
   // 
   //  mode_Alm_H_MaskOn     MODE — Masks the high alarm             Bool    
   //                    (1 = alarm masked, 0 = normal)
   //  mode_Alm_L_MaskOn     MODE — Masks the low alarm            Bool    
   //                    (1 = alarm masked, 0 = normal)
   //  mode_Wrn_H_MaskOn     MODE — Masks the high warning            Bool    
   //                    (1 = warning masked, 0 = normal)
   //  mode_Wrn_L_MaskOn      MODE — Masks the low warning                 Bool    
   //                    (1 = warning masked, 0 = normal)
   //  mode_SimOn         MODE — Simulation mode               Bool
   //                    (1 = sim mode active, 0 = normal)
   //  mode_SimValue       MODE — Simulation value               Real
   //                    (engineering units)
   //  mode_LocalOn         MODE — Local HMI control enabled           Bool
   //                    (1 = active, 0 = disabled or N/A)
   //  mode_RemoteOn        MODE — Remote SCADA control enabled       Bool
   //                    (1 = active, 0 = disabled or N/A)
   // 
   //  msg_Alm_H         MESSAGE — Alarm - high alarm is active        Bool
   //  msg_Alm_L          MESSAGE — Alarm - low alarm is active          Bool
   //  msg_Wrn_H          MESSAGE — Warning - high warning is active      Bool
   //  msg_Wrn_L          MESSAGE — Warning - low warning is active        Bool
   //  msg_Flt_External         MESSAGE — Fault - external fault signal is active      Bool
   //  msg_Flt_OverRange¹     MESSAGE — Fault - instrument is over-range       Bool
   //  msg_Flt_UnderRange¹      MESSAGE — Fault - instrument is under-range       Bool
   //  msg_Flt_OutOfRange¹      MESSAGE — Fault - instrument is out-of-range        Bool
   // 
   //  batch_ID         BATCH — Booking ID (optional for batch operations)   Int
   // 
   //  actual_Value          ACTUAL — SCALED INSTRUMENT VALUE         Real
   //                      [engineering units]
   //  actual_Alm_H_Timer      ACTUAL — Timer value — alarm high operation     Real
   //                      timer [seconds]
   //  actual_Alm_L_Timer       ACTUAL — Timer value — alarm low operation    Real
   //                      timer [seconds]
   //  actual_Wrn_H_Timer      ACTUAL — Timer value — warning high operation    Real
   //                      timer [seconds]
   //  actual_Wrn_L_Timer       ACTUAL — Timer value — warning low operation      Real
   //                      timer [seconds]
   // 
   //  $pret_AlmHEn           INTERNAL — Edge retention (+ve) alarm high en      Bool
   //  $Pret_AlmLEn            INTERNAL — Edge retention (+ve) alarm low en     Bool
   //  $pret_WrnHEn           INTERNAL — Edge retention (+ve) warning high en     Bool
   //  $pret_WrnLEn            INTERNAL — Edge retention (+ve) warning low en       Bool
   //  ――――――――――――――――――――――――――――――――――――――――――
   //  ¹        msg_Flt_OverRange, msg_Flt_UnderRange and msg_Flt_OutOfRange will all
   //      activate if a configuration error is active status_ConfigError = 1, actual_Value will 
   //      also be set to zero under these conditions.
   // 
   // With the exception of the flowing, all these signals are discussed in the previous sections, the 
   // outstanding items are firstly:
   // 
   //      batch_ID
   // 
   // The batch_ID is not required for normal use; it is only used where a “booking” system is used 
   // (common in batch and routing applications). Such booking applications can acquire the device 
   // if it is free and reserve it for a particular phase of the batch. Batch applications are a topic in 
   // their own right and are discussed separately in the online User Guide.
   // 
   // Next:
   //      actual_Alm_H_Timer	Real
   //      actual_Alm_L_Timer	Real
   //      actual_Wrn_H_Timer	Real
   //      actual_Wrn_L_Timer	Real
   // 
   // These data points hold the actual value of the running timer for each of the alarms/warnings, 
   // both on and off-delay timers used the same timer within the block (the timers are mutually 
   // exclusive, only one will be running at once for each alarm or warning — hence only one timer is
   // needed for each alarm or warning).
   // 
   // Each timer counts down from the TIME_ values (UT02001_St_InstAnalogRead) to zero in 200 ms
   // intervals.
   // 
   // Finally:
   //      $pret_AlmHEn
   //      $Pret_AlmLEn
   //      $pret_WrnHEn
   //      $pret_WrnLEn
   // 
   // These are internal working signals (all signals the start with a $ are internal working signals 
   // used by the block). In this instance they are used to detect a rising edge on each of the alarm 
   // and warning enable signals. 
   // 
   //                ━━━   ⬙⬙⬙⬙⬙⬙   ━━━
   // 
   // 
   // 
   // ▄▄▄▄▄▄▄▄▄▄▄▄▄▄▄▄▄▄▄▄▄▄▄▄▄▄▄▄▄▄▄▄▄▄▄▄▄▄▄▄▄▄▄▄
   // 6.     CONSTANTS AND TEMPORARY (LOCAL) DATA
   // 
   // 
   // The following constants and temporary data storage are used:
   // 
   // 
   //  Temporary (local) data
   //  ――――――――――――――――――――――――――――――――――――――――――
   //  SIGNAL NAME          FUNCTION                  TYPE
   //  ――――――――――――――――――――――――――――――――――――――――――
   //  revInfo             Revision information for the block         UT01000
   //  licInfo           Licensing information for the block      UT01001
   //  wrkAlmHEn          Working Alm_H is enabled and not masked   Bool
   //  wrkAlmLEn        Working Alm_L is enabled and not masked    Bool
   //  wrkWrnHEn           Working Wrn_H is enabled and not masked    Bool
   //  wrkWrnLEn           Working Wrn_L is enabled and not masked    Bool
   //  calcPart1           Scale value part 1 (RAW_ANALOG − RAW_MIN)   Real
   //  calcPart2           Scale value part 2 (SCALE_MAX − SCALE_MIN)   Real
   //  calcPart3           Scale value part 3 (RAW_MAX − RAW_MIN)     Real
   //  calcRawOOR        Calculated OOR absolute value          Real
   //  calcOverRange       Calculated over range limit (in raw units)    Real
   //  calcUnderRange       Calculated under range limit (in raw units)     Real
   //  calcHystAbs         Absolute hysteresis value           Real
   //  wrkHyst           Working hysteresis value            Real
   //  wrkOORPercent         Working out of range percentage          Real
   //  wrkInt           Working storage area (integer)          Int
   //  wrkReal           Working storage (Real)             Real
   //  wrkDInt           Working storage area (double integer)         DInt
   //  ――――――――――――――――――――――――――――――――――――――――――
   // 
   //                ━━━   ⬙⬙⬙⬙⬙⬙   ━━━
   // 
   // 
   // 
   // ▄▄▄▄▄▄▄▄▄▄▄▄▄▄▄▄▄▄▄▄▄▄▄▄▄▄▄▄▄▄▄▄▄▄▄▄▄▄▄▄▄▄▄▄
   // 7.     BLOCK CALLS
   // 
   // There are no PAL block calls from within this block.
   // 
   //                ━━━   ⬙⬙⬙⬙⬙⬙   ━━━
   // 
   // 
   // 
   // ▄▄▄▄▄▄▄▄▄▄▄▄▄▄▄▄▄▄▄▄▄▄▄▄▄▄▄▄▄▄▄▄▄▄▄▄▄▄▄▄▄▄▄▄
   // 8.     ASSOCIATED BLOCKS
   // 
   // 
   // This is a stand-alone block and is not associated with any other blocks.
   // 
   //                ━━━   ⬙⬙⬙⬙⬙⬙   ━━━
   // 
   // 
   // 
   // ▄▄▄▄▄▄▄▄▄▄▄▄▄▄▄▄▄▄▄▄▄▄▄▄▄▄▄▄▄▄▄▄▄▄▄▄▄▄▄▄▄▄▄▄
   // 9.     SYSTEM BLOCK CALLS AND SYSTEM DATA TYPES
   // 
   // There are no system block calls.
   // 
   //                ━━━   ⬙⬙⬙⬙⬙⬙   ━━━
   // 
   // 
   // 
   // ▄▄▄▄▄▄▄▄▄▄▄▄▄▄▄▄▄▄▄▄▄▄▄▄▄▄▄▄▄▄▄▄▄▄▄▄▄▄▄▄▄▄▄▄
   // 10.     SPECIAL PROPERTIES AND REQUIREMENTS
   // 
   // 
   // 
   // ▂▂▂▂▂▂▂▂▂▂▂▂▂▂▂▂▂▂▂▂▂▂▂▂▂▂▂▂▂▂▂▂▂▂▂▂▂▂▂▂▂▂▂▂
   // 10.1   Block optimisation
   // 
   // 
   // Block optimisation is ACTIVE for this block
   // 
   // 
   // 
   // ▂▂▂▂▂▂▂▂▂▂▂▂▂▂▂▂▂▂▂▂▂▂▂▂▂▂▂▂▂▂▂▂▂▂▂▂▂▂▂▂▂▂▂▂
   // 10.2   Calling requirements
   // 
   // 
   // There are no special calling requirements for this block.
   // 
   //                ━━━   ⬙⬙⬙⬙⬙⬙   ━━━
   // 
   // 
   // 
   // ▄▄▄▄▄▄▄▄▄▄▄▄▄▄▄▄▄▄▄▄▄▄▄▄▄▄▄▄▄▄▄▄▄▄▄▄▄▄▄▄▄▄▄▄
   // 11.     EXAMPLE USAGE
   // 
   // 
   // The following shows a typical deployment of FC02001:
   // 
   //                         ┌─────────────
   //      ───────────────────┤ FC02001 
   //                         ├───────────────┤
   //    "DB21001_DY_StdGlobalData".SysSignals ─┤ SYS_SIGNALS
   //                         │               │
   //                          "FC001" ─┤ RAW_ANALOG           │
   //                         │               │
   //           "FC001_FAULT"           │               │
   //        ────┤╱├──────────┤ EXT_FAULT                │
   //                         │               │
   //                         │               │
   //     "DB02001_St_StdInstAnalogRead".FC001 ─┤ STATIC_DATA             │
   //                         │
   //     "DB22001_Dy_StdInstAnalogRead".FC001 ─┤ DYNAMIC_DATA
   //                         │
   //                         │
   //                                         │
   //                                ─────────┘
   // 
   // 
   //               ━━━   ⬙⬙⬙⬙⬙⬙   ━━━
   // 
   // 
   // 
   // ██████████████ █ █ █ █  END   █ █ █ █ ██████████████
END_REGION

REGION Network 4: Current revision and modification history
   // ▄▄▄▄▄▄▄▄▄▄▄▄▄▄▄▄▄▄▄▄▄▄▄▄▄▄▄▄▄▄▄▄▄▄▄▄▄▄▄▄▄▄▄▄
   // MODIFICATION HISTORY
   // 
   // 
   // The revision data shown here, in the network comments, contains additional information 
   // reflecting the software development workflow under the version control system (VCS) employed 
   // to track all software changes.
   // 
   // The VCS in use is the Git Source Code Management system in conjunction with the GitHub online 
   // hosting system. The software in its entirety is available in the GitHub remote repository:
   // 
   //      https://github.com/practicalseries/PS2001-pal-software
   // 
   // The repository is public and can be freely copied (forked in GitHub terminology) and used 
   // under the MIT licence. 
   // 
   // The MIT licence is reproduced in full in the last network of this software module
   // 
   // 
   //  ―――――――――――――――――――――――――――――――――――――――――――
   //  DATE       REVISION            MASTER BRANCH      DEV
   //          (nnn.amm)   COMMIT TAG    (Base ---> Merge)    BRANCH   Author
   //  ———————————————————————————————————————————
   //  2021.02.18    001.000   D0002A-001.000   D0002 N/A     D0002B   M. Gledhill
   //                        FC02001 Migration to VCS — Released for test
   // 
   //  2021.02.18    000.801   D0002A-000.801   D0002 N/A     D0002B   M. Gledhill
   //                        FC02001 Migration to VCS — Released for test
   //  ———————————————————————————————————————————
   //   Where: nnn  =  Major revision
   //         a  =  Type (1-7 Development, 8 Proving, 9 Qualification, 0 Release)
   //       mm  =  Minor revision (must be 00 if a = 0)
   //         Block properties version number should be set to nn.a (only one decimal place)
   // 
   // ▄▄▄▄▄▄▄▄▄▄▄▄▄▄▄▄▄▄▄▄▄▄▄▄▄▄▄▄▄▄▄▄▄▄▄▄▄▄▄▄▄▄▄▄
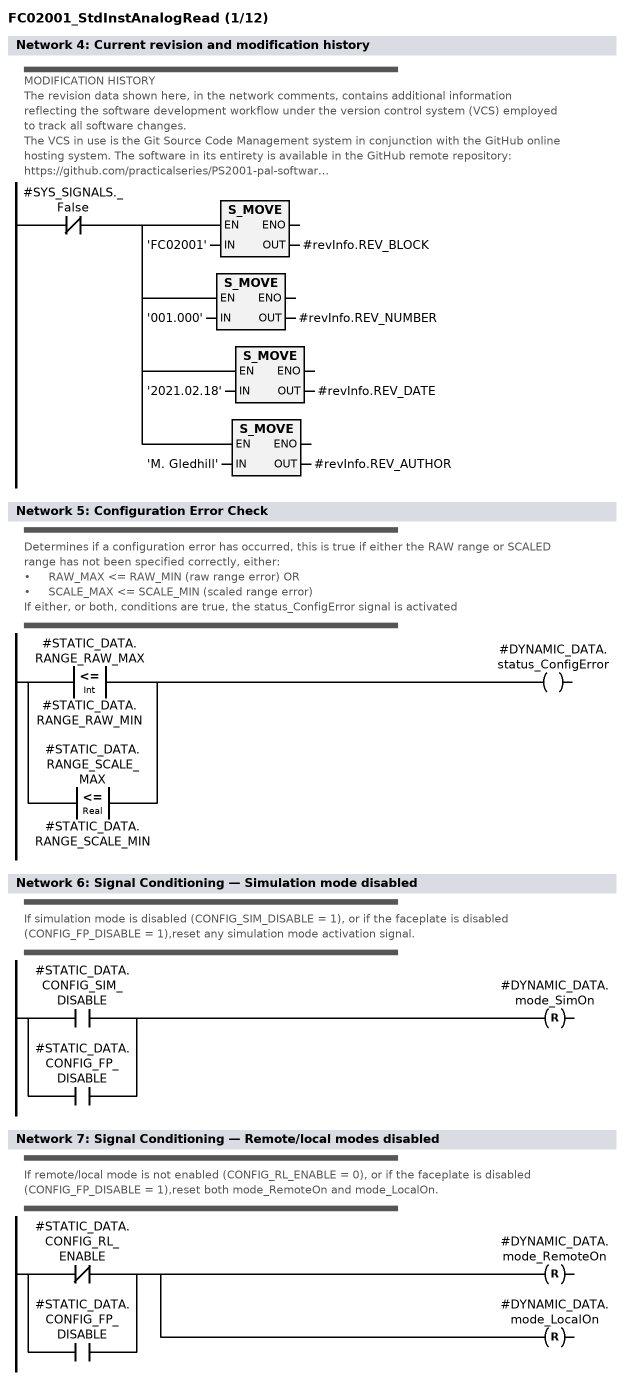
   RUNG wire#powerrail
      I_Contact( #SYS_SIGNALS._False )
      wire#w1
      S_Move(in := 'FC02001', out => #revInfo.REV_BLOCK)
   END_RUNG
   RUNG wire#w1
      S_Move(in := '001.000', out => #revInfo.REV_NUMBER)
   END_RUNG
   RUNG wire#w1
      S_Move(in := '2021.02.18', out => #revInfo.REV_DATE)
   END_RUNG
   RUNG wire#w1
      S_Move(in := 'M. Gledhill', out => #revInfo.REV_AUTHOR)
   END_RUNG
   // the same network as SCL:
   IF NOT #SYS_SIGNALS._False THEN
       #revInfo.REV_BLOCK := 'FC02001';
       #revInfo.REV_NUMBER := '001.000';
       #revInfo.REV_DATE := '2021.02.18';
       #revInfo.REV_AUTHOR := 'M. Gledhill';
   END_IF;
END_REGION

REGION Network 5: Configuration Error Check
   // ▀▀▀▀▀▀▀▀▀▀▀▀▀▀▀▀▀▀▀▀▀▀▀▀▀▀▀▀▀▀▀▀▀▀▀▀▀▀▀▀▀▀▀▀
   // 
   // Determines if a configuration error has occurred, this is true if either the RAW range or SCALED 
   // range has not been specified correctly, either:
   // 
   //    •   RAW_MAX <= RAW_MIN (raw range error) OR
   //    •   SCALE_MAX <= SCALE_MIN (scaled range error)
   // 
   // If either, or both, conditions are true, the status_ConfigError signal is activated
   // ▄▄▄▄▄▄▄▄▄▄▄▄▄▄▄▄▄▄▄▄▄▄▄▄▄▄▄▄▄▄▄▄▄▄▄▄▄▄▄▄▄▄▄▄
   RUNG wire#powerrail
      { S7_Templates := "SrcType := Int" } LE_Contact(in1 := #STATIC_DATA.RANGE_RAW_MAX, in2 := #STATIC_DATA.RANGE_RAW_MIN)
      wire#w1
      Coil( #DYNAMIC_DATA.status_ConfigError )
   END_RUNG
   RUNG wire#powerrail
      { S7_Templates := "SrcType := Real" } LE_Contact(in1 := #STATIC_DATA.RANGE_SCALE_MAX, in2 := #STATIC_DATA.RANGE_SCALE_MIN)
   END_RUNG wire#w1
   // the same network as SCL:
   #DYNAMIC_DATA.status_ConfigError := (#STATIC_DATA.RANGE_RAW_MAX <= #STATIC_DATA.RANGE_RAW_MIN) OR (#STATIC_DATA.RANGE_SCALE_MAX <= #STATIC_DATA.RANGE_SCALE_MIN);
END_REGION

REGION Network 6: Signal Conditioning — Simulation mode disabled
   // ▀▀▀▀▀▀▀▀▀▀▀▀▀▀▀▀▀▀▀▀▀▀▀▀▀▀▀▀▀▀▀▀▀▀▀▀▀▀▀▀▀▀▀▀
   // If simulation mode is disabled (CONFIG_SIM_DISABLE = 1), or if the faceplate is disabled 
   // (CONFIG_FP_DISABLE = 1),reset any simulation mode activation signal.
   // ▄▄▄▄▄▄▄▄▄▄▄▄▄▄▄▄▄▄▄▄▄▄▄▄▄▄▄▄▄▄▄▄▄▄▄▄▄▄▄▄▄▄▄▄
   RUNG wire#powerrail
      Contact( #STATIC_DATA.CONFIG_SIM_DISABLE )
      wire#w1
      R_Coil( #DYNAMIC_DATA.mode_SimOn )
   END_RUNG
   RUNG wire#powerrail
      Contact( #STATIC_DATA.CONFIG_FP_DISABLE )
   END_RUNG wire#w1
   // the same network as SCL:
   IF #STATIC_DATA.CONFIG_SIM_DISABLE OR #STATIC_DATA.CONFIG_FP_DISABLE THEN
       #DYNAMIC_DATA.mode_SimOn := FALSE;
   END_IF;
END_REGION

REGION Network 7: Signal Conditioning — Remote/local modes disabled
   // ▀▀▀▀▀▀▀▀▀▀▀▀▀▀▀▀▀▀▀▀▀▀▀▀▀▀▀▀▀▀▀▀▀▀▀▀▀▀▀▀▀▀▀▀
   // If remote/local mode is not enabled (CONFIG_RL_ENABLE = 0), or if the faceplate is disabled 
   // (CONFIG_FP_DISABLE = 1),reset both mode_RemoteOn and mode_LocalOn.
   // ▄▄▄▄▄▄▄▄▄▄▄▄▄▄▄▄▄▄▄▄▄▄▄▄▄▄▄▄▄▄▄▄▄▄▄▄▄▄▄▄▄▄▄▄
   RUNG wire#powerrail
      I_Contact( #STATIC_DATA.CONFIG_RL_ENABLE )
      wire#w1
      R_Coil( #DYNAMIC_DATA.mode_RemoteOn )
   END_RUNG
   RUNG wire#powerrail
      Contact( #STATIC_DATA.CONFIG_FP_DISABLE )
   END_RUNG wire#w1
   RUNG wire#w1
      R_Coil( #DYNAMIC_DATA.mode_LocalOn )
   END_RUNG
   // the same network as SCL:
   IF NOT #STATIC_DATA.CONFIG_RL_ENABLE OR #STATIC_DATA.CONFIG_FP_DISABLE THEN
       #DYNAMIC_DATA.mode_RemoteOn := FALSE;
       #DYNAMIC_DATA.mode_LocalOn := FALSE;
   END_IF;
END_REGION

REGION Network 8: Signal Conditioning — Remote/Local selection if enabled
   // ▀▀▀▀▀▀▀▀▀▀▀▀▀▀▀▀▀▀▀▀▀▀▀▀▀▀▀▀▀▀▀▀▀▀▀▀▀▀▀▀▀▀▀▀
   // If remote/local mode is enabled (CONFIG_RL_ENABLE = 1), and the  faceplate is not disabled 
   // (CONFIG_FP_DISABLE = 0), and:
   // 
   //    1.  Neither mode_RemoteOn or mode_LocalOn is active, default to remote mode
   //    2.  A rising edge is detected on mode_LocalOn, reset mode_RemoteOn (in local)
   //    3.  A rising edge is detected on mode_RemoteOn, reset mode_LocalOn (in remote)
   //    4.  Both mode_RemoteOn and mode_LocalOn is active, default to remote mode
   // ▄▄▄▄▄▄▄▄▄▄▄▄▄▄▄▄▄▄▄▄▄▄▄▄▄▄▄▄▄▄▄▄▄▄▄▄▄▄▄▄▄▄▄▄
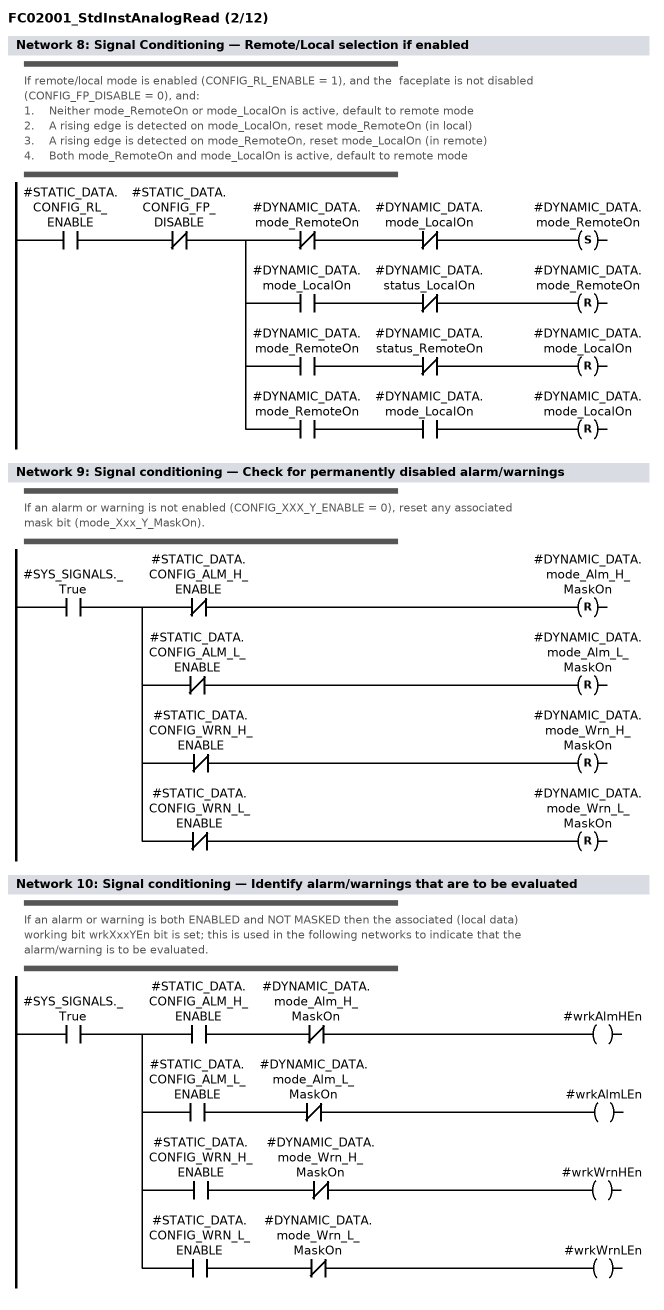
   RUNG wire#powerrail
      Contact( #STATIC_DATA.CONFIG_RL_ENABLE )
      I_Contact( #STATIC_DATA.CONFIG_FP_DISABLE )
      wire#w1
      I_Contact( #DYNAMIC_DATA.mode_RemoteOn )
      I_Contact( #DYNAMIC_DATA.mode_LocalOn )
      S_Coil( #DYNAMIC_DATA.mode_RemoteOn )
   END_RUNG
   RUNG wire#w1
      Contact( #DYNAMIC_DATA.mode_LocalOn )
      I_Contact( #DYNAMIC_DATA.status_LocalOn )
      R_Coil( #DYNAMIC_DATA.mode_RemoteOn )
   END_RUNG
   RUNG wire#w1
      Contact( #DYNAMIC_DATA.mode_RemoteOn )
      I_Contact( #DYNAMIC_DATA.status_RemoteOn )
      R_Coil( #DYNAMIC_DATA.mode_LocalOn )
   END_RUNG
   RUNG wire#w1
      Contact( #DYNAMIC_DATA.mode_RemoteOn )
      Contact( #DYNAMIC_DATA.mode_LocalOn )
      R_Coil( #DYNAMIC_DATA.mode_LocalOn )
   END_RUNG
   // the same network as SCL:
   #_w1 := #STATIC_DATA.CONFIG_RL_ENABLE AND NOT #STATIC_DATA.CONFIG_FP_DISABLE;
   IF #_w1 AND NOT #DYNAMIC_DATA.mode_RemoteOn AND NOT #DYNAMIC_DATA.mode_LocalOn THEN
       #DYNAMIC_DATA.mode_RemoteOn := TRUE;
   END_IF;
   IF #_w1 AND #DYNAMIC_DATA.mode_LocalOn AND NOT #DYNAMIC_DATA.status_LocalOn THEN
       #DYNAMIC_DATA.mode_RemoteOn := FALSE;
   END_IF;
   IF #_w1 AND #DYNAMIC_DATA.mode_RemoteOn AND NOT #DYNAMIC_DATA.status_RemoteOn THEN
       #DYNAMIC_DATA.mode_LocalOn := FALSE;
   END_IF;
   IF #_w1 AND #DYNAMIC_DATA.mode_RemoteOn AND #DYNAMIC_DATA.mode_LocalOn THEN
       #DYNAMIC_DATA.mode_LocalOn := FALSE;
   END_IF;
END_REGION

REGION Network 9: Signal conditioning — Check for permanently disabled alarm/warnings
   // ▀▀▀▀▀▀▀▀▀▀▀▀▀▀▀▀▀▀▀▀▀▀▀▀▀▀▀▀▀▀▀▀▀▀▀▀▀▀▀▀▀▀▀▀
   // If an alarm or warning is not enabled (CONFIG_XXX_Y_ENABLE = 0), reset any associated 
   // mask bit (mode_Xxx_Y_MaskOn).
   // ▄▄▄▄▄▄▄▄▄▄▄▄▄▄▄▄▄▄▄▄▄▄▄▄▄▄▄▄▄▄▄▄▄▄▄▄▄▄▄▄▄▄▄▄
   RUNG wire#powerrail
      Contact( #SYS_SIGNALS._True )
      wire#w1
      I_Contact( #STATIC_DATA.CONFIG_ALM_H_ENABLE )
      R_Coil( #DYNAMIC_DATA.mode_Alm_H_MaskOn )
   END_RUNG
   RUNG wire#w1
      I_Contact( #STATIC_DATA.CONFIG_ALM_L_ENABLE )
      R_Coil( #DYNAMIC_DATA.mode_Alm_L_MaskOn )
   END_RUNG
   RUNG wire#w1
      I_Contact( #STATIC_DATA.CONFIG_WRN_H_ENABLE )
      R_Coil( #DYNAMIC_DATA.mode_Wrn_H_MaskOn )
   END_RUNG
   RUNG wire#w1
      I_Contact( #STATIC_DATA.CONFIG_WRN_L_ENABLE )
      R_Coil( #DYNAMIC_DATA.mode_Wrn_L_MaskOn )
   END_RUNG
   // the same network as SCL:
   IF #SYS_SIGNALS._True AND NOT #STATIC_DATA.CONFIG_ALM_H_ENABLE THEN
       #DYNAMIC_DATA.mode_Alm_H_MaskOn := FALSE;
   END_IF;
   IF #SYS_SIGNALS._True AND NOT #STATIC_DATA.CONFIG_ALM_L_ENABLE THEN
       #DYNAMIC_DATA.mode_Alm_L_MaskOn := FALSE;
   END_IF;
   IF #SYS_SIGNALS._True AND NOT #STATIC_DATA.CONFIG_WRN_H_ENABLE THEN
       #DYNAMIC_DATA.mode_Wrn_H_MaskOn := FALSE;
   END_IF;
   IF #SYS_SIGNALS._True AND NOT #STATIC_DATA.CONFIG_WRN_L_ENABLE THEN
       #DYNAMIC_DATA.mode_Wrn_L_MaskOn := FALSE;
   END_IF;
END_REGION

REGION Network 10: Signal conditioning — Identify alarm/warnings that are to be evaluated
   // ▀▀▀▀▀▀▀▀▀▀▀▀▀▀▀▀▀▀▀▀▀▀▀▀▀▀▀▀▀▀▀▀▀▀▀▀▀▀▀▀▀▀▀▀
   // If an alarm or warning is both ENABLED and NOT MASKED then the associated (local data) 
   // working bit wrkXxxYEn bit is set; this is used in the following networks to indicate that the 
   // alarm/warning is to be evaluated.
   // ▄▄▄▄▄▄▄▄▄▄▄▄▄▄▄▄▄▄▄▄▄▄▄▄▄▄▄▄▄▄▄▄▄▄▄▄▄▄▄▄▄▄▄▄
   RUNG wire#powerrail
      Contact( #SYS_SIGNALS._True )
      wire#w1
      Contact( #STATIC_DATA.CONFIG_ALM_H_ENABLE )
      I_Contact( #DYNAMIC_DATA.mode_Alm_H_MaskOn )
      Coil( #wrkAlmHEn )
   END_RUNG
   RUNG wire#w1
      Contact( #STATIC_DATA.CONFIG_ALM_L_ENABLE )
      I_Contact( #DYNAMIC_DATA.mode_Alm_L_MaskOn )
      Coil( #wrkAlmLEn )
   END_RUNG
   RUNG wire#w1
      Contact( #STATIC_DATA.CONFIG_WRN_H_ENABLE )
      I_Contact( #DYNAMIC_DATA.mode_Wrn_H_MaskOn )
      Coil( #wrkWrnHEn )
   END_RUNG
   RUNG wire#w1
      Contact( #STATIC_DATA.CONFIG_WRN_L_ENABLE )
      I_Contact( #DYNAMIC_DATA.mode_Wrn_L_MaskOn )
      Coil( #wrkWrnLEn )
   END_RUNG
   // the same network as SCL:
   #wrkAlmHEn := #SYS_SIGNALS._True AND #STATIC_DATA.CONFIG_ALM_H_ENABLE AND NOT #DYNAMIC_DATA.mode_Alm_H_MaskOn;
   #wrkAlmLEn := #SYS_SIGNALS._True AND #STATIC_DATA.CONFIG_ALM_L_ENABLE AND NOT #DYNAMIC_DATA.mode_Alm_L_MaskOn;
   #wrkWrnHEn := #SYS_SIGNALS._True AND #STATIC_DATA.CONFIG_WRN_H_ENABLE AND NOT #DYNAMIC_DATA.mode_Wrn_H_MaskOn;
   #wrkWrnLEn := #SYS_SIGNALS._True AND #STATIC_DATA.CONFIG_WRN_L_ENABLE AND NOT #DYNAMIC_DATA.mode_Wrn_L_MaskOn;
END_REGION

REGION Network 11: Signal conditioning — Reset the data for alarm/warnings that are not enabled
   // ▀▀▀▀▀▀▀▀▀▀▀▀▀▀▀▀▀▀▀▀▀▀▀▀▀▀▀▀▀▀▀▀▀▀▀▀▀▀▀▀▀▀▀▀
   // If an alarm or warning is not enabled or is masked (indicated by wrkXxxYEn = 0), the associated 
   // message bit (msg_Xxx_Y) for the alarm or warning is permanently deactivated (reset).
   // 
   // Similarly, the associated actual timer for the alarm or warning (actual_Xxx_Y_Timer) is set to 
   // zero.
   // ▄▄▄▄▄▄▄▄▄▄▄▄▄▄▄▄▄▄▄▄▄▄▄▄▄▄▄▄▄▄▄▄▄▄▄▄▄▄▄▄▄▄▄▄
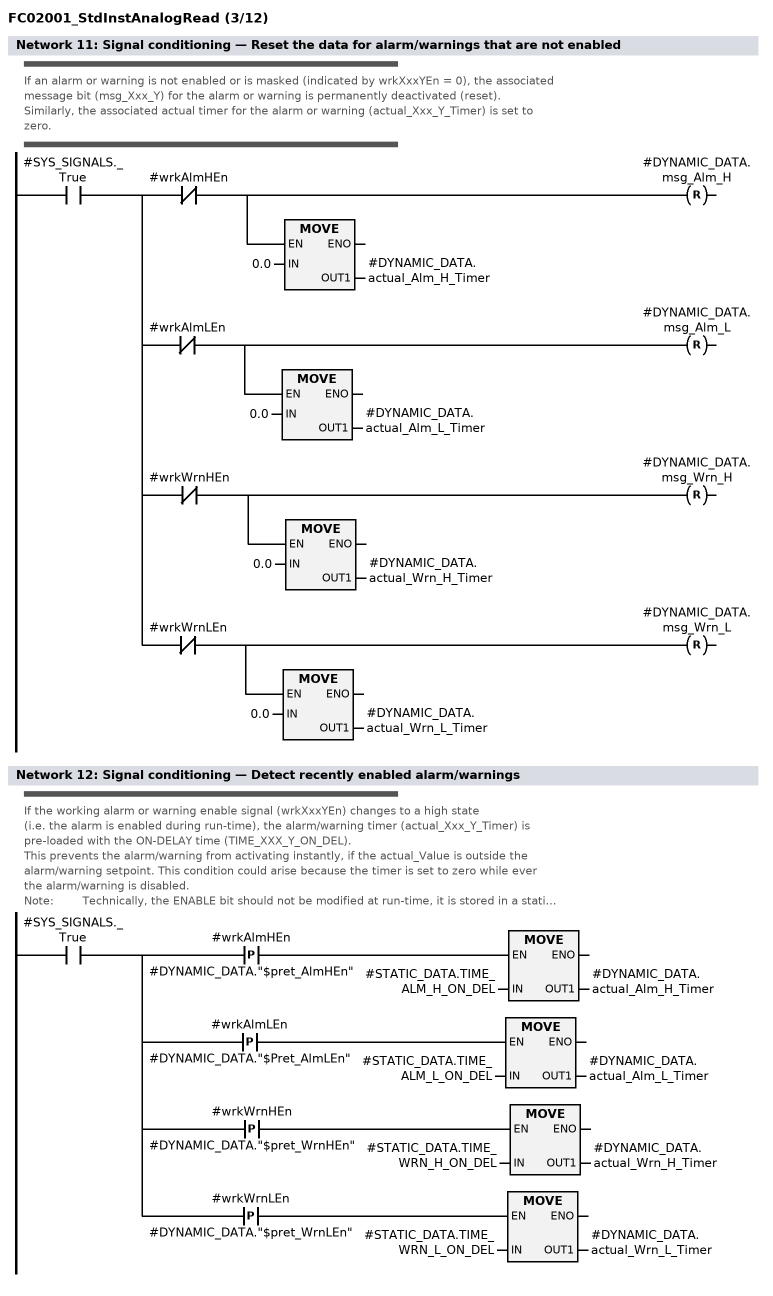
   RUNG wire#powerrail
      Contact( #SYS_SIGNALS._True )
      wire#w1
      I_Contact( #wrkAlmHEn )
      wire#w2
      R_Coil( #DYNAMIC_DATA.msg_Alm_H )
   END_RUNG
   RUNG wire#w2
      { S7_GenerateENO := "TRUE" } Move(in := 0.0, out1 => #DYNAMIC_DATA.actual_Alm_H_Timer)
   END_RUNG
   RUNG wire#w1
      I_Contact( #wrkAlmLEn )
      wire#w3
      R_Coil( #DYNAMIC_DATA.msg_Alm_L )
   END_RUNG
   RUNG wire#w3
      { S7_GenerateENO := "TRUE" } Move(in := 0.0, out1 => #DYNAMIC_DATA.actual_Alm_L_Timer)
   END_RUNG
   RUNG wire#w1
      I_Contact( #wrkWrnHEn )
      wire#w4
      R_Coil( #DYNAMIC_DATA.msg_Wrn_H )
   END_RUNG
   RUNG wire#w4
      { S7_GenerateENO := "TRUE" } Move(in := 0.0, out1 => #DYNAMIC_DATA.actual_Wrn_H_Timer)
   END_RUNG
   RUNG wire#w1
      I_Contact( #wrkWrnLEn )
      wire#w5
      R_Coil( #DYNAMIC_DATA.msg_Wrn_L )
   END_RUNG
   RUNG wire#w5
      { S7_GenerateENO := "TRUE" } Move(in := 0.0, out1 => #DYNAMIC_DATA.actual_Wrn_L_Timer)
   END_RUNG
   // the same network as SCL:
   IF #SYS_SIGNALS._True AND NOT #wrkAlmHEn THEN
       #DYNAMIC_DATA.msg_Alm_H := FALSE;
       #DYNAMIC_DATA.actual_Alm_H_Timer := 0.0;
   END_IF;
   IF #SYS_SIGNALS._True AND NOT #wrkAlmLEn THEN
       #DYNAMIC_DATA.msg_Alm_L := FALSE;
       #DYNAMIC_DATA.actual_Alm_L_Timer := 0.0;
   END_IF;
   IF #SYS_SIGNALS._True AND NOT #wrkWrnHEn THEN
       #DYNAMIC_DATA.msg_Wrn_H := FALSE;
       #DYNAMIC_DATA.actual_Wrn_H_Timer := 0.0;
   END_IF;
   IF #SYS_SIGNALS._True AND NOT #wrkWrnLEn THEN
       #DYNAMIC_DATA.msg_Wrn_L := FALSE;
       #DYNAMIC_DATA.actual_Wrn_L_Timer := 0.0;
   END_IF;
END_REGION

REGION Network 12: Signal conditioning — Detect recently enabled alarm/warnings
   // ▀▀▀▀▀▀▀▀▀▀▀▀▀▀▀▀▀▀▀▀▀▀▀▀▀▀▀▀▀▀▀▀▀▀▀▀▀▀▀▀▀▀▀▀
   // If the working alarm or warning enable signal (wrkXxxYEn) changes to a high state
   // (i.e. the alarm is enabled during run-time), the alarm/warning timer (actual_Xxx_Y_Timer) is 
   // pre-loaded with the ON-DELAY time (TIME_XXX_Y_ON_DEL).
   // 
   // This prevents the alarm/warning from activating instantly, if the actual_Value is outside the
   // alarm/warning setpoint. This condition could arise because the timer is set to zero while ever
   // the alarm/warning is disabled.
   // 
   // Note:    Technically, the ENABLE bit should not be modified at run-time, it is stored in a static
   //      data block; however, the condition could arise if that static data block is being used
   //      as a recipe block. mask signals can of course be changed at run-time.
   // ▄▄▄▄▄▄▄▄▄▄▄▄▄▄▄▄▄▄▄▄▄▄▄▄▄▄▄▄▄▄▄▄▄▄▄▄▄▄▄▄▄▄▄▄
   RUNG wire#powerrail
      Contact( #SYS_SIGNALS._True )
      wire#w1
      P_Contact(operand := #wrkAlmHEn, bit := #DYNAMIC_DATA."$pret_AlmHEn")
      { S7_GenerateENO := "TRUE" } Move(in := #STATIC_DATA.TIME_ALM_H_ON_DEL, out1 => #DYNAMIC_DATA.actual_Alm_H_Timer)
   END_RUNG
   RUNG wire#w1
      P_Contact(operand := #wrkAlmLEn, bit := #DYNAMIC_DATA."$Pret_AlmLEn")
      { S7_GenerateENO := "TRUE" } Move(in := #STATIC_DATA.TIME_ALM_L_ON_DEL, out1 => #DYNAMIC_DATA.actual_Alm_L_Timer)
   END_RUNG
   RUNG wire#w1
      P_Contact(operand := #wrkWrnHEn, bit := #DYNAMIC_DATA."$pret_WrnHEn")
      { S7_GenerateENO := "TRUE" } Move(in := #STATIC_DATA.TIME_WRN_H_ON_DEL, out1 => #DYNAMIC_DATA.actual_Wrn_H_Timer)
   END_RUNG
   RUNG wire#w1
      P_Contact(operand := #wrkWrnLEn, bit := #DYNAMIC_DATA."$pret_WrnLEn")
      { S7_GenerateENO := "TRUE" } Move(in := #STATIC_DATA.TIME_WRN_L_ON_DEL, out1 => #DYNAMIC_DATA.actual_Wrn_L_Timer)
   END_RUNG
   // the same network as SCL:
   #_w1 := #SYS_SIGNALS._True AND #wrkAlmHEn AND NOT #DYNAMIC_DATA."$pret_AlmHEn";   // rising edge of #wrkAlmHEn
   #DYNAMIC_DATA."$pret_AlmHEn" := #wrkAlmHEn;
   IF #_w1 THEN #DYNAMIC_DATA.actual_Alm_H_Timer := #STATIC_DATA.TIME_ALM_H_ON_DEL; END_IF;
   #_w2 := #SYS_SIGNALS._True AND #wrkAlmLEn AND NOT #DYNAMIC_DATA."$Pret_AlmLEn";   // rising edge of #wrkAlmLEn
   #DYNAMIC_DATA."$Pret_AlmLEn" := #wrkAlmLEn;
   IF #_w2 THEN #DYNAMIC_DATA.actual_Alm_L_Timer := #STATIC_DATA.TIME_ALM_L_ON_DEL; END_IF;
   #_w3 := #SYS_SIGNALS._True AND #wrkWrnHEn AND NOT #DYNAMIC_DATA."$pret_WrnHEn";   // rising edge of #wrkWrnHEn
   #DYNAMIC_DATA."$pret_WrnHEn" := #wrkWrnHEn;
   IF #_w3 THEN #DYNAMIC_DATA.actual_Wrn_H_Timer := #STATIC_DATA.TIME_WRN_H_ON_DEL; END_IF;
   #_w4 := #SYS_SIGNALS._True AND #wrkWrnLEn AND NOT #DYNAMIC_DATA."$pret_WrnLEn";   // rising edge of #wrkWrnLEn
   #DYNAMIC_DATA."$pret_WrnLEn" := #wrkWrnLEn;
   IF #_w4 THEN #DYNAMIC_DATA.actual_Wrn_L_Timer := #STATIC_DATA.TIME_WRN_L_ON_DEL; END_IF;
END_REGION

REGION Network 13: Signal conditioning — Ensure Out of Range percentage is 10% or less
   // ▀▀▀▀▀▀▀▀▀▀▀▀▀▀▀▀▀▀▀▀▀▀▀▀▀▀▀▀▀▀▀▀▀▀▀▀▀▀▀▀▀▀▀▀
   // The RANGE_OOR_PERCENT signal is checked to ensure it is within the range 0.0 to 10.0.
   // 
   // The local data wrkOORPercent holds the corrected value and is used in the out of range 
   // calculations
   // ▄▄▄▄▄▄▄▄▄▄▄▄▄▄▄▄▄▄▄▄▄▄▄▄▄▄▄▄▄▄▄▄▄▄▄▄▄▄▄▄▄▄▄▄
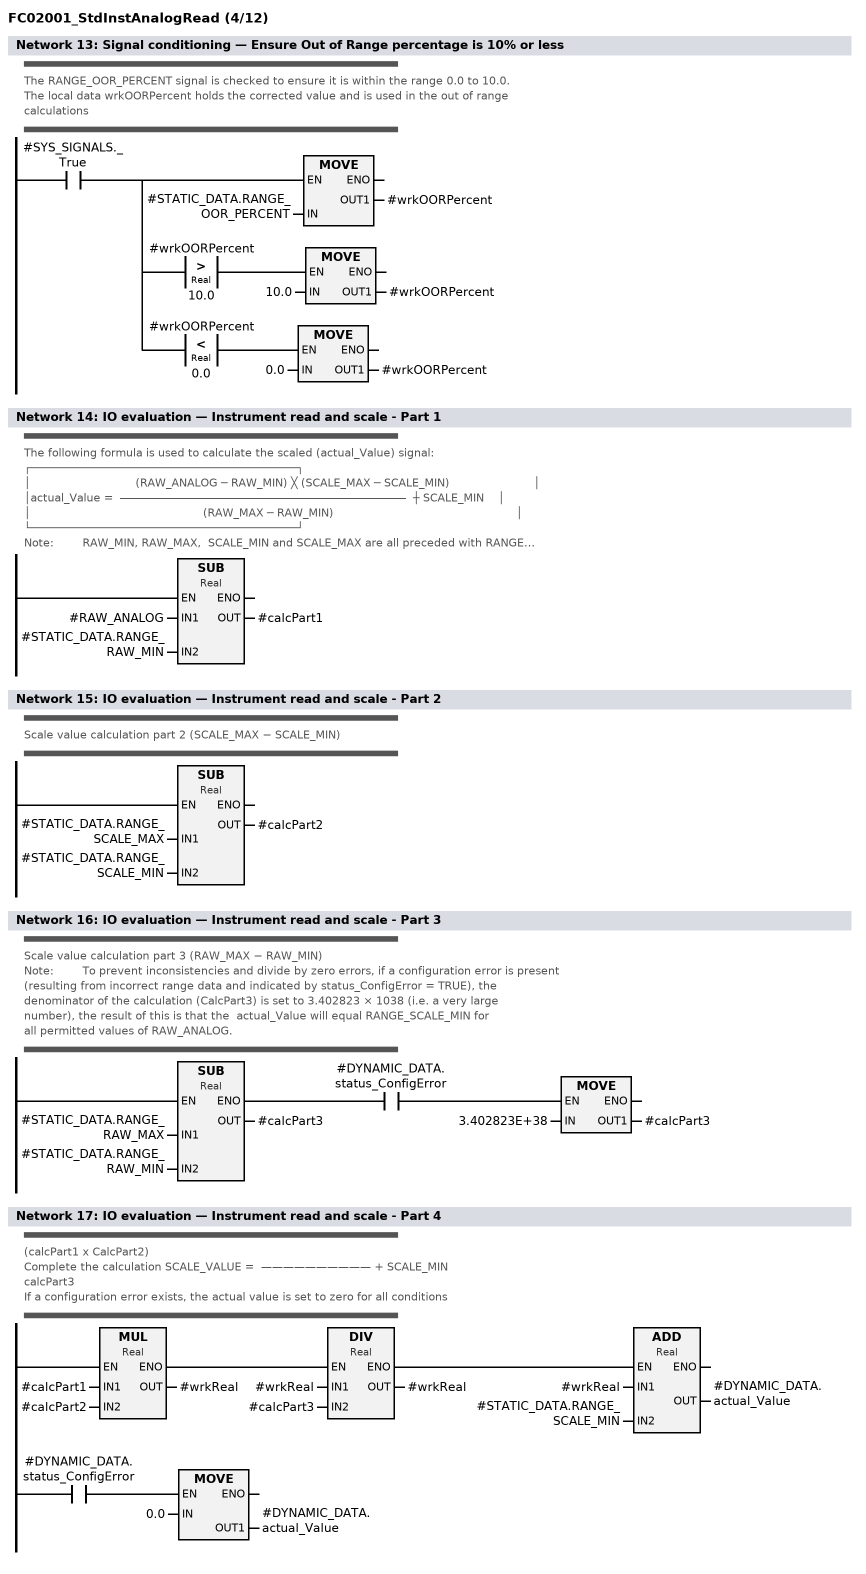
   RUNG wire#powerrail
      Contact( #SYS_SIGNALS._True )
      wire#w1
      { S7_GenerateENO := "TRUE" } Move(in := #STATIC_DATA.RANGE_OOR_PERCENT, out1 => #wrkOORPercent)
   END_RUNG
   RUNG wire#w1
      { S7_Templates := "SrcType := Real" } GT_Contact(in1 := #wrkOORPercent, in2 := 10.0)
      { S7_GenerateENO := "TRUE" } Move(in := 10.0, out1 => #wrkOORPercent)
   END_RUNG
   RUNG wire#w1
      { S7_Templates := "SrcType := Real" } LT_Contact(in1 := #wrkOORPercent, in2 := 0.0)
      { S7_GenerateENO := "TRUE" } Move(in := 0.0, out1 => #wrkOORPercent)
   END_RUNG
   // the same network as SCL:
   IF #SYS_SIGNALS._True THEN #wrkOORPercent := #STATIC_DATA.RANGE_OOR_PERCENT; END_IF;
   IF #SYS_SIGNALS._True AND (#wrkOORPercent > 10.0) THEN #wrkOORPercent := 10.0; END_IF;
   IF #SYS_SIGNALS._True AND (#wrkOORPercent < 0.0) THEN #wrkOORPercent := 0.0; END_IF;
END_REGION

REGION Network 14: IO evaluation — Instrument read and scale - Part 1
   // ▀▀▀▀▀▀▀▀▀▀▀▀▀▀▀▀▀▀▀▀▀▀▀▀▀▀▀▀▀▀▀▀▀▀▀▀▀▀▀▀▀▀▀▀
   // The following formula is used to calculate the scaled (actual_Value) signal:
   // ┌─────────────────────────────────────────┐
   // │                              (RAW_ANALOG ─ RAW_MIN) ╳ (SCALE_MAX ─ SCALE_MIN)            │
   // │actual_Value =  ――――――――――――――――――――――――――  ┼ SCALE_MIN    │
   // │                              (RAW_MAX ─ RAW_MIN)                    │
   // └─────────────────────────────────────────┘
   // Note:    RAW_MIN, RAW_MAX,  SCALE_MIN and SCALE_MAX are all preceded with RANGE_
   //      in the above equation 
   // 
   // Scale value calculation part 1 is (RAW_ANALOG − RAW_MIN)
   // ▄▄▄▄▄▄▄▄▄▄▄▄▄▄▄▄▄▄▄▄▄▄▄▄▄▄▄▄▄▄▄▄▄▄▄▄▄▄▄▄▄▄▄▄
   RUNG wire#powerrail
      { S7_Templates := "SrcType := Real"; S7_GenerateENO := "TRUE" } Sub(in1 := #RAW_ANALOG, in2 := #STATIC_DATA.RANGE_RAW_MIN, out => #calcPart1)
   END_RUNG
   // the same network as SCL:
   #calcPart1 := #RAW_ANALOG - #STATIC_DATA.RANGE_RAW_MIN;
END_REGION

REGION Network 15: IO evaluation — Instrument read and scale - Part 2
   // ▀▀▀▀▀▀▀▀▀▀▀▀▀▀▀▀▀▀▀▀▀▀▀▀▀▀▀▀▀▀▀▀▀▀▀▀▀▀▀▀▀▀▀▀
   // Scale value calculation part 2 (SCALE_MAX − SCALE_MIN)
   // ▄▄▄▄▄▄▄▄▄▄▄▄▄▄▄▄▄▄▄▄▄▄▄▄▄▄▄▄▄▄▄▄▄▄▄▄▄▄▄▄▄▄▄▄
   RUNG wire#powerrail
      { S7_Templates := "SrcType := Real"; S7_GenerateENO := "TRUE" } Sub(in1 := #STATIC_DATA.RANGE_SCALE_MAX, in2 := #STATIC_DATA.RANGE_SCALE_MIN, out => #calcPart2)
   END_RUNG
   // the same network as SCL:
   #calcPart2 := #STATIC_DATA.RANGE_SCALE_MAX - #STATIC_DATA.RANGE_SCALE_MIN;
END_REGION

REGION Network 16: IO evaluation — Instrument read and scale - Part 3
   // ▀▀▀▀▀▀▀▀▀▀▀▀▀▀▀▀▀▀▀▀▀▀▀▀▀▀▀▀▀▀▀▀▀▀▀▀▀▀▀▀▀▀▀▀
   // Scale value calculation part 3 (RAW_MAX − RAW_MIN)
   // 
   // Note:    To prevent inconsistencies and divide by zero errors, if a configuration error is present
   //      (resulting from incorrect range data and indicated by status_ConfigError = TRUE), the
   //      denominator of the calculation (CalcPart3) is set to 3.402823 × 1038 (i.e. a very large 
   //      number), the result of this is that the  actual_Value will equal RANGE_SCALE_MIN for 
   //      all permitted values of RAW_ANALOG.
   // ▄▄▄▄▄▄▄▄▄▄▄▄▄▄▄▄▄▄▄▄▄▄▄▄▄▄▄▄▄▄▄▄▄▄▄▄▄▄▄▄▄▄▄▄
   RUNG wire#powerrail
      { S7_Templates := "SrcType := Real"; S7_GenerateENO := "TRUE" } Sub(in1 := #STATIC_DATA.RANGE_RAW_MAX, in2 := #STATIC_DATA.RANGE_RAW_MIN, out => #calcPart3)
      Contact( #DYNAMIC_DATA.status_ConfigError )
      Move(in := 3.402823E+38, out1 => #calcPart3)
   END_RUNG
   // the same network as SCL:
   // ENO of a box is taken as its EN; it also drops when the box reports an error
   #calcPart3 := #STATIC_DATA.RANGE_RAW_MAX - #STATIC_DATA.RANGE_RAW_MIN;
   IF #DYNAMIC_DATA.status_ConfigError THEN #calcPart3 := 3.402823E+38; END_IF;
END_REGION

REGION Network 17: IO evaluation — Instrument read and scale - Part 4
   // ▀▀▀▀▀▀▀▀▀▀▀▀▀▀▀▀▀▀▀▀▀▀▀▀▀▀▀▀▀▀▀▀▀▀▀▀▀▀▀▀▀▀▀▀
   //                                                                              (calcPart1 x CalcPart2)
   // Complete the calculation SCALE_VALUE =  —————————— + SCALE_MIN
   //                                                                                         calcPart3
   // 
   // If a configuration error exists, the actual value is set to zero for all conditions
   // ▄▄▄▄▄▄▄▄▄▄▄▄▄▄▄▄▄▄▄▄▄▄▄▄▄▄▄▄▄▄▄▄▄▄▄▄▄▄▄▄▄▄▄▄
   RUNG wire#powerrail
      { S7_Templates := "SrcType := Real"; S7_GenerateENO := "TRUE" } Mul(in1 := #calcPart1, in2 := #calcPart2, out => #wrkReal)
      { S7_Templates := "SrcType := Real"; S7_GenerateENO := "TRUE" } Div(in1 := #wrkReal, in2 := #calcPart3, out => #wrkReal)
      { S7_Templates := "SrcType := Real"; S7_GenerateENO := "TRUE" } Add(in1 := #wrkReal, in2 := #STATIC_DATA.RANGE_SCALE_MIN, out => #DYNAMIC_DATA.actual_Value)
   END_RUNG
   RUNG wire#powerrail
      Contact( #DYNAMIC_DATA.status_ConfigError )
      Move(in := 0.0, out1 => #DYNAMIC_DATA.actual_Value)
   END_RUNG
   // the same network as SCL:
   // ENO of a box is taken as its EN; it also drops when the box reports an error
   #wrkReal := #calcPart1 * #calcPart2;
   #wrkReal := #wrkReal / #calcPart3;
   #DYNAMIC_DATA.actual_Value := #wrkReal + #STATIC_DATA.RANGE_SCALE_MIN;
   IF #DYNAMIC_DATA.status_ConfigError THEN #DYNAMIC_DATA.actual_Value := 0.0; END_IF;
END_REGION

REGION Network 18: IO evaluation — Calculate out of range value
   // ▀▀▀▀▀▀▀▀▀▀▀▀▀▀▀▀▀▀▀▀▀▀▀▀▀▀▀▀▀▀▀▀▀▀▀▀▀▀▀▀▀▀▀▀
   // The out of range limits are calculated from the raw span of the instrument 
   // (RAW_MAX - RAW_MIN, stored in calcPart3).
   // 
   // The absolute value of the out of range tolerance is stored in calcRawOOR and is calculated as
   // follows:
   // 
   // 
   //                                (RAW_MAX - RAW_MIN) x wrkOORPercent
   // calcRawOOR  =  ————————————————————
   //                                                                100
   // 
   // OR
   // 
   //                               calcPart3 x wrkOORPercent
   // calcRawOOR  =  ——————————————
   //                                                 100
   // 
   // 
   // The instrument is over range if the RAW_ANALOG is greater than RAW_MAX + calcRawOOR
   // 
   // The instrument is under range if the RAW_ANALOG is less than RAW_MIN - calcRawOOR
   // ▄▄▄▄▄▄▄▄▄▄▄▄▄▄▄▄▄▄▄▄▄▄▄▄▄▄▄▄▄▄▄▄▄▄▄▄▄▄▄▄▄▄▄▄
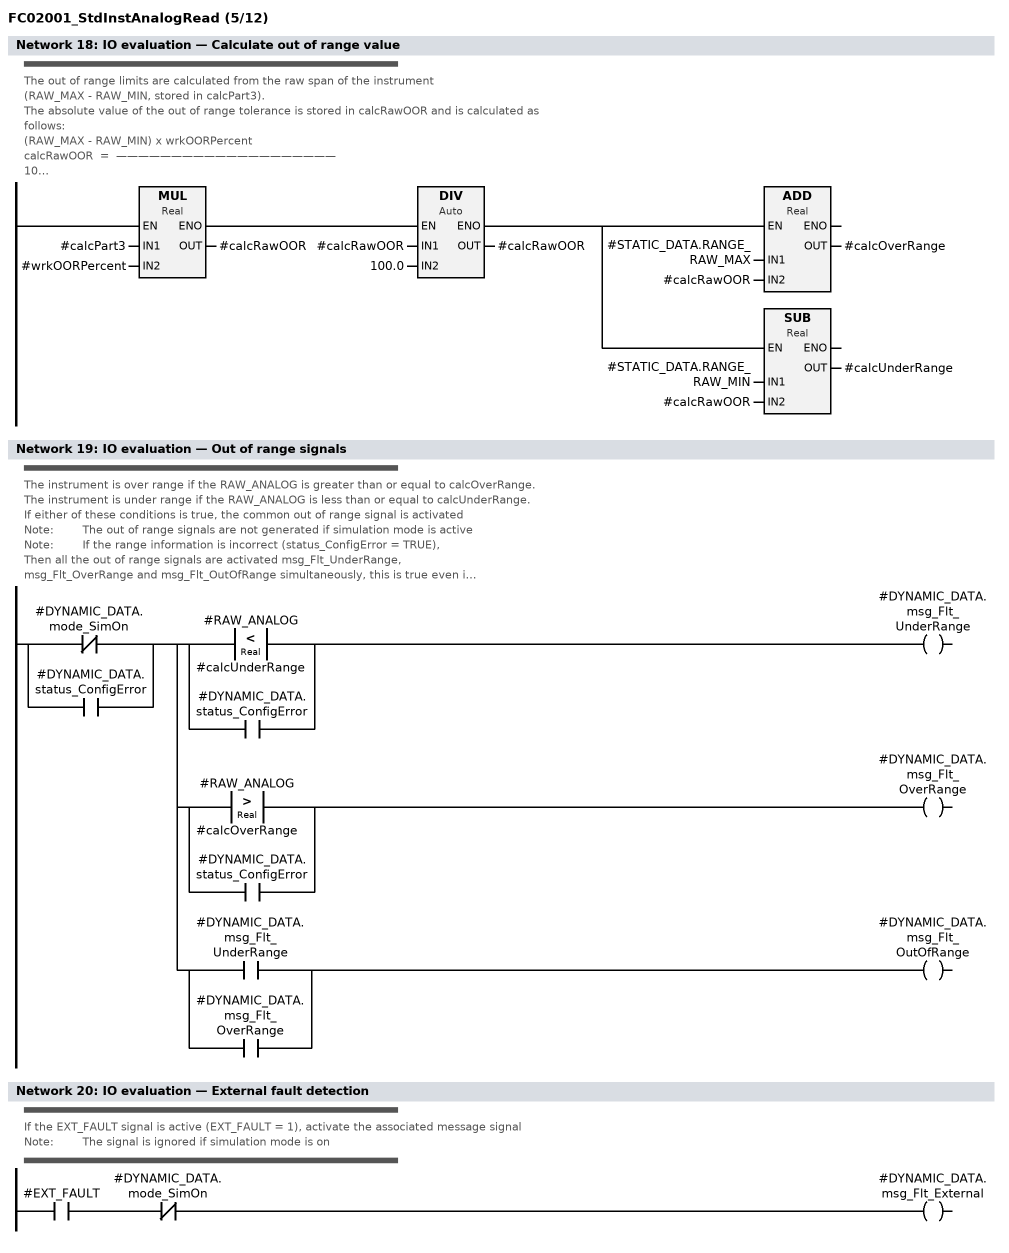
   RUNG wire#powerrail
      { S7_Templates := "SrcType := Real"; S7_GenerateENO := "TRUE" } Mul(in1 := #calcPart3, in2 := #wrkOORPercent, out => #calcRawOOR)
      Div(in1 := #calcRawOOR, in2 := 100.0, out => #calcRawOOR)
      wire#w1
      { S7_Templates := "SrcType := Real"; S7_GenerateENO := "TRUE" } Add(in1 := #STATIC_DATA.RANGE_RAW_MAX, in2 := #calcRawOOR, out => #calcOverRange)
   END_RUNG
   RUNG wire#w1
      { S7_Templates := "SrcType := Real"; S7_GenerateENO := "TRUE" } Sub(in1 := #STATIC_DATA.RANGE_RAW_MIN, in2 := #calcRawOOR, out => #calcUnderRange)
   END_RUNG
   // the same network as SCL:
   // ENO of a box is taken as its EN; it also drops when the box reports an error
   #calcRawOOR := #calcPart3 * #wrkOORPercent;
   #calcRawOOR := #calcRawOOR / 100.0;
   #calcOverRange := #STATIC_DATA.RANGE_RAW_MAX + #calcRawOOR;
   #calcUnderRange := #STATIC_DATA.RANGE_RAW_MIN - #calcRawOOR;
END_REGION

REGION Network 19: IO evaluation — Out of range signals
   // ▀▀▀▀▀▀▀▀▀▀▀▀▀▀▀▀▀▀▀▀▀▀▀▀▀▀▀▀▀▀▀▀▀▀▀▀▀▀▀▀▀▀▀▀
   // The instrument is over range if the RAW_ANALOG is greater than or equal to calcOverRange.
   // 
   // The instrument is under range if the RAW_ANALOG is less than or equal to calcUnderRange.
   // 
   // If either of these conditions is true, the common out of range signal is activated
   // 
   // Note:    The out of range signals are not generated if simulation mode is active
   // 
   // Note:    If the range information is incorrect (status_ConfigError = TRUE),
   //      Then all the out of range signals are activated msg_Flt_UnderRange, 
   //      msg_Flt_OverRange and msg_Flt_OutOfRange simultaneously, this is true even if
   //      simulation mode is active.
   // ▄▄▄▄▄▄▄▄▄▄▄▄▄▄▄▄▄▄▄▄▄▄▄▄▄▄▄▄▄▄▄▄▄▄▄▄▄▄▄▄▄▄▄▄
   RUNG wire#powerrail
      I_Contact( #DYNAMIC_DATA.mode_SimOn )
      wire#w1
      { S7_Templates := "SrcType := Real" } LT_Contact(in1 := #RAW_ANALOG, in2 := #calcUnderRange)
      wire#w2
      Coil( #DYNAMIC_DATA.msg_Flt_UnderRange )
   END_RUNG
   RUNG wire#powerrail
      Contact( #DYNAMIC_DATA.status_ConfigError )
   END_RUNG wire#w1
   RUNG wire#w1
      Contact( #DYNAMIC_DATA.status_ConfigError )
   END_RUNG wire#w2
   RUNG wire#w1
      { S7_Templates := "SrcType := Real" } GT_Contact(in1 := #RAW_ANALOG, in2 := #calcOverRange)
      wire#w3
      Coil( #DYNAMIC_DATA.msg_Flt_OverRange )
   END_RUNG
   RUNG wire#w1
      Contact( #DYNAMIC_DATA.status_ConfigError )
   END_RUNG wire#w3
   RUNG wire#w1
      Contact( #DYNAMIC_DATA.msg_Flt_UnderRange )
      wire#w4
      Coil( #DYNAMIC_DATA.msg_Flt_OutOfRange )
   END_RUNG
   RUNG wire#w1
      Contact( #DYNAMIC_DATA.msg_Flt_OverRange )
   END_RUNG wire#w4
   // the same network as SCL:
   #_w1 := NOT #DYNAMIC_DATA.mode_SimOn OR #DYNAMIC_DATA.status_ConfigError;
   #DYNAMIC_DATA.msg_Flt_UnderRange := #_w1 AND ((#RAW_ANALOG < #calcUnderRange) OR #DYNAMIC_DATA.status_ConfigError);
   #DYNAMIC_DATA.msg_Flt_OverRange := #_w1 AND ((#RAW_ANALOG > #calcOverRange) OR #DYNAMIC_DATA.status_ConfigError);
   #DYNAMIC_DATA.msg_Flt_OutOfRange := #_w1 AND (#DYNAMIC_DATA.msg_Flt_UnderRange OR #DYNAMIC_DATA.msg_Flt_OverRange);
END_REGION

REGION Network 20: IO evaluation — External fault detection
   // ▀▀▀▀▀▀▀▀▀▀▀▀▀▀▀▀▀▀▀▀▀▀▀▀▀▀▀▀▀▀▀▀▀▀▀▀▀▀▀▀▀▀▀▀
   // If the EXT_FAULT signal is active (EXT_FAULT = 1), activate the associated message signal
   // 
   // Note:    The signal is ignored if simulation mode is on
   // ▄▄▄▄▄▄▄▄▄▄▄▄▄▄▄▄▄▄▄▄▄▄▄▄▄▄▄▄▄▄▄▄▄▄▄▄▄▄▄▄▄▄▄▄
   RUNG wire#powerrail
      Contact( #EXT_FAULT )
      I_Contact( #DYNAMIC_DATA.mode_SimOn )
      Coil( #DYNAMIC_DATA.msg_Flt_External )
   END_RUNG
   // the same network as SCL:
   #DYNAMIC_DATA.msg_Flt_External := #EXT_FAULT AND NOT #DYNAMIC_DATA.mode_SimOn;
END_REGION

REGION Network 21: Operating mode — Simulation mode
   // ▀▀▀▀▀▀▀▀▀▀▀▀▀▀▀▀▀▀▀▀▀▀▀▀▀▀▀▀▀▀▀▀▀▀▀▀▀▀▀▀▀▀▀▀
   // If simulation mode is enabled (mode_SimOn = 1) and a configuration error is not present,
   // (status_ConfigError = 0) overwrite the actual_Value with the mode_SimValue signal set by the 
   // operator.
   // 
   // Note:    Any fault signals will be suppressed (turned off) is simulation mode is active
   //      and a configuration error is not present
   // 
   //      The simulated value (mode_SimValue) is restricted to the range given in 
   //      RANGE_SCALE_MIN and RANGE_SCALE_MAX
   // ▄▄▄▄▄▄▄▄▄▄▄▄▄▄▄▄▄▄▄▄▄▄▄▄▄▄▄▄▄▄▄▄▄▄▄▄▄▄▄▄▄▄▄▄
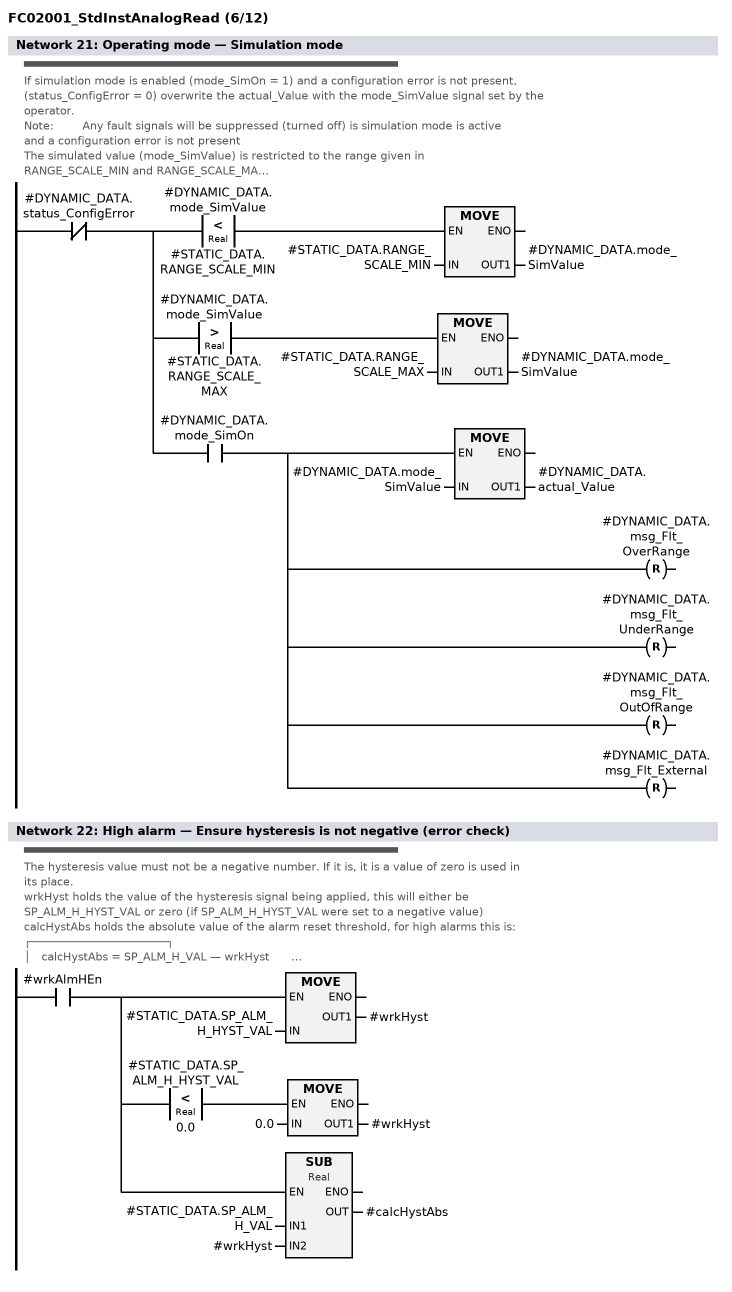
   RUNG wire#powerrail
      I_Contact( #DYNAMIC_DATA.status_ConfigError )
      wire#w1
      { S7_Templates := "SrcType := Real" } LT_Contact(in1 := #DYNAMIC_DATA.mode_SimValue, in2 := #STATIC_DATA.RANGE_SCALE_MIN)
      { S7_GenerateENO := "TRUE" } Move(in := #STATIC_DATA.RANGE_SCALE_MIN, out1 => #DYNAMIC_DATA.mode_SimValue)
   END_RUNG
   RUNG wire#w1
      { S7_Templates := "SrcType := Real" } GT_Contact(in1 := #DYNAMIC_DATA.mode_SimValue, in2 := #STATIC_DATA.RANGE_SCALE_MAX)
      { S7_GenerateENO := "TRUE" } Move(in := #STATIC_DATA.RANGE_SCALE_MAX, out1 => #DYNAMIC_DATA.mode_SimValue)
   END_RUNG
   RUNG wire#w1
      Contact( #DYNAMIC_DATA.mode_SimOn )
      wire#w2
      { S7_GenerateENO := "TRUE" } Move(in := #DYNAMIC_DATA.mode_SimValue, out1 => #DYNAMIC_DATA.actual_Value)
   END_RUNG
   RUNG wire#w2
      R_Coil( #DYNAMIC_DATA.msg_Flt_OverRange )
   END_RUNG
   RUNG wire#w2
      R_Coil( #DYNAMIC_DATA.msg_Flt_UnderRange )
   END_RUNG
   RUNG wire#w2
      R_Coil( #DYNAMIC_DATA.msg_Flt_OutOfRange )
   END_RUNG
   RUNG wire#w2
      R_Coil( #DYNAMIC_DATA.msg_Flt_External )
   END_RUNG
   // the same network as SCL:
   #_w1 := NOT #DYNAMIC_DATA.status_ConfigError;
   IF #_w1 AND (#DYNAMIC_DATA.mode_SimValue < #STATIC_DATA.RANGE_SCALE_MIN) THEN
       #DYNAMIC_DATA.mode_SimValue := #STATIC_DATA.RANGE_SCALE_MIN;
   END_IF;
   IF #_w1 AND (#DYNAMIC_DATA.mode_SimValue > #STATIC_DATA.RANGE_SCALE_MAX) THEN
       #DYNAMIC_DATA.mode_SimValue := #STATIC_DATA.RANGE_SCALE_MAX;
   END_IF;
   IF #_w1 AND #DYNAMIC_DATA.mode_SimOn THEN
       #DYNAMIC_DATA.actual_Value := #DYNAMIC_DATA.mode_SimValue;
       #DYNAMIC_DATA.msg_Flt_OverRange := FALSE;
       #DYNAMIC_DATA.msg_Flt_UnderRange := FALSE;
       #DYNAMIC_DATA.msg_Flt_OutOfRange := FALSE;
       #DYNAMIC_DATA.msg_Flt_External := FALSE;
   END_IF;
END_REGION

REGION Network 22: High alarm — Ensure hysteresis is not negative (error check)
   // ▀▀▀▀▀▀▀▀▀▀▀▀▀▀▀▀▀▀▀▀▀▀▀▀▀▀▀▀▀▀▀▀▀▀▀▀▀▀▀▀▀▀▀▀
   // The hysteresis value must not be a negative number. If it is, it is a value of zero is used in
   // its place.
   // 
   // wrkHyst holds the value of the hysteresis signal being applied, this will either be 
   // SP_ALM_H_HYST_VAL or zero (if SP_ALM_H_HYST_VAL were set to a negative value)
   // 
   // calcHystAbs holds the absolute value of the alarm reset threshold, for high alarms this is:
   // ┌─────────────────────┐
   // │ calcHystAbs = SP_ALM_H_VAL — wrkHyst    │
   // └─────────────────────┘
   // 
   // The two threshold values for the high alarm are thus:
   // 
   //      High alarm activation threshold = SP_ALM_H_VAL
   //      High alarm reset threshold          = calcHystAbs
   // 
   // Note:    The hysteresis is only checked if alarm is being evaluated
   // ▄▄▄▄▄▄▄▄▄▄▄▄▄▄▄▄▄▄▄▄▄▄▄▄▄▄▄▄▄▄▄▄▄▄▄▄▄▄▄▄▄▄▄▄
   RUNG wire#powerrail
      Contact( #wrkAlmHEn )
      wire#w1
      { S7_GenerateENO := "TRUE" } Move(in := #STATIC_DATA.SP_ALM_H_HYST_VAL, out1 => #wrkHyst)
   END_RUNG
   RUNG wire#w1
      { S7_Templates := "SrcType := Real" } LT_Contact(in1 := #STATIC_DATA.SP_ALM_H_HYST_VAL, in2 := 0.0)
      { S7_GenerateENO := "TRUE" } Move(in := 0.0, out1 => #wrkHyst)
   END_RUNG
   RUNG wire#w1
      { S7_Templates := "SrcType := Real"; S7_GenerateENO := "TRUE" } Sub(in1 := #STATIC_DATA.SP_ALM_H_VAL, in2 := #wrkHyst, out => #calcHystAbs)
   END_RUNG
   // the same network as SCL:
   IF #wrkAlmHEn THEN #wrkHyst := #STATIC_DATA.SP_ALM_H_HYST_VAL; END_IF;
   IF #wrkAlmHEn AND (#STATIC_DATA.SP_ALM_H_HYST_VAL < 0.0) THEN #wrkHyst := 0.0; END_IF;
   IF #wrkAlmHEn THEN #calcHystAbs := #STATIC_DATA.SP_ALM_H_VAL - #wrkHyst; END_IF;
END_REGION

REGION Network 23: High alarm — Check for activation level and ON-DELAY timer
   // ▀▀▀▀▀▀▀▀▀▀▀▀▀▀▀▀▀▀▀▀▀▀▀▀▀▀▀▀▀▀▀▀▀▀▀▀▀▀▀▀▀▀▀▀
   // If the high alarm has been enabled and is not masked and the actual_Value is greater than or 
   // equal to the alarm setpoint (SP_ALM_H_VAL), but the alarm has not yet been triggered 
   // (msg_Alm_H = 0) then the ON-DELAY phase is active (the alarm timer is counting down).
   // 
   // The timer will begin to count down from the value in TIME_ALM_H_ON_DEL using the 200ms 
   // pulse (it will count down in increments of 0.2s). If the high alarm timer is less than or equal to 
   // zero, then the ON-DELAY has expired and the High Alarm message will become active.
   // 
   // If at any point during the ON-DELAY count down, the actual_Value drops below the activation
   // setpoint (SP_ALM_H_VAL), the timer will be reset to the TIME_ALM_H_ON_DEL value, forcing 
   // the ON-DELAY to start again.
   // ▄▄▄▄▄▄▄▄▄▄▄▄▄▄▄▄▄▄▄▄▄▄▄▄▄▄▄▄▄▄▄▄▄▄▄▄▄▄▄▄▄▄▄▄
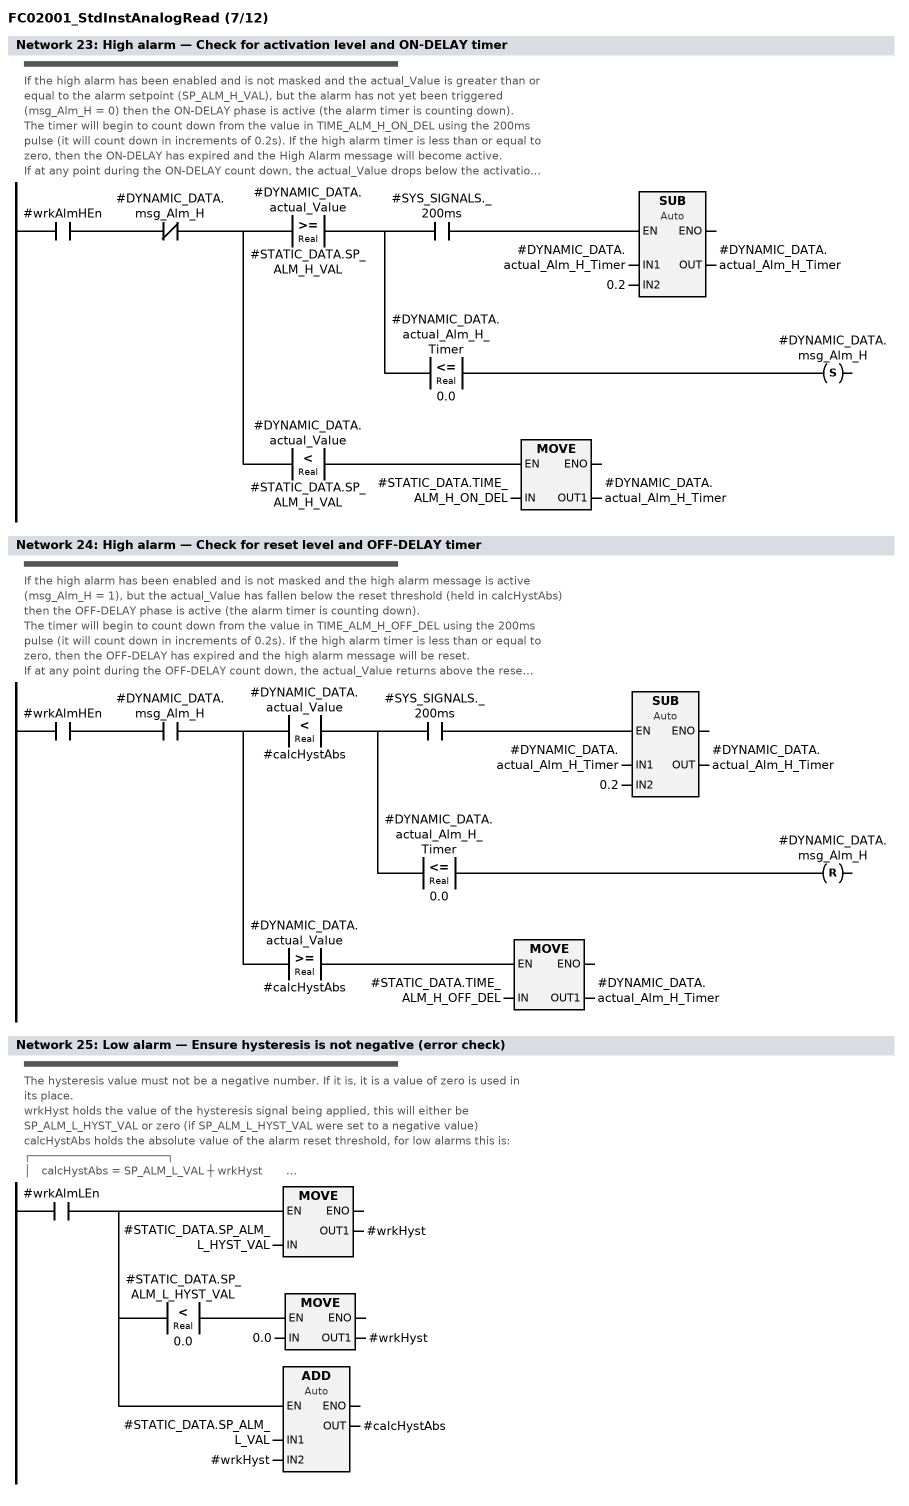
   RUNG wire#powerrail
      Contact( #wrkAlmHEn )
      I_Contact( #DYNAMIC_DATA.msg_Alm_H )
      wire#w1
      { S7_Templates := "SrcType := Real" } GE_Contact(in1 := #DYNAMIC_DATA.actual_Value, in2 := #STATIC_DATA.SP_ALM_H_VAL)
      wire#w2
      Contact( #SYS_SIGNALS._200ms )
      Sub(in1 := #DYNAMIC_DATA.actual_Alm_H_Timer, in2 := 0.2, out => #DYNAMIC_DATA.actual_Alm_H_Timer)
   END_RUNG
   RUNG wire#w2
      { S7_Templates := "SrcType := Real" } LE_Contact(in1 := #DYNAMIC_DATA.actual_Alm_H_Timer, in2 := 0.0)
      S_Coil( #DYNAMIC_DATA.msg_Alm_H )
   END_RUNG
   RUNG wire#w1
      { S7_Templates := "SrcType := Real" } LT_Contact(in1 := #DYNAMIC_DATA.actual_Value, in2 := #STATIC_DATA.SP_ALM_H_VAL)
      { S7_GenerateENO := "TRUE" } Move(in := #STATIC_DATA.TIME_ALM_H_ON_DEL, out1 => #DYNAMIC_DATA.actual_Alm_H_Timer)
   END_RUNG
   // the same network as SCL:
   #_w1 := #wrkAlmHEn AND NOT #DYNAMIC_DATA.msg_Alm_H;
   #_w2 := #_w1 AND (#DYNAMIC_DATA.actual_Value >= #STATIC_DATA.SP_ALM_H_VAL);
   IF #_w2 AND #SYS_SIGNALS._200ms THEN
       #DYNAMIC_DATA.actual_Alm_H_Timer := #DYNAMIC_DATA.actual_Alm_H_Timer - 0.2;
   END_IF;
   IF #_w2 AND (#DYNAMIC_DATA.actual_Alm_H_Timer <= 0.0) THEN #DYNAMIC_DATA.msg_Alm_H := TRUE; END_IF;
   IF #_w1 AND (#DYNAMIC_DATA.actual_Value < #STATIC_DATA.SP_ALM_H_VAL) THEN
       #DYNAMIC_DATA.actual_Alm_H_Timer := #STATIC_DATA.TIME_ALM_H_ON_DEL;
   END_IF;
END_REGION

REGION Network 24: High alarm — Check for reset level and OFF-DELAY timer
   // ▀▀▀▀▀▀▀▀▀▀▀▀▀▀▀▀▀▀▀▀▀▀▀▀▀▀▀▀▀▀▀▀▀▀▀▀▀▀▀▀▀▀▀▀
   // If the high alarm has been enabled and is not masked and the high alarm message is active 
   // (msg_Alm_H = 1), but the actual_Value has fallen below the reset threshold (held in calcHystAbs) 
   // then the OFF-DELAY phase is active (the alarm timer is counting down).
   // 
   // The timer will begin to count down from the value in TIME_ALM_H_OFF_DEL using the 200ms 
   // pulse (it will count down in increments of 0.2s). If the high alarm timer is less than or equal to 
   // zero, then the OFF-DELAY has expired and the high alarm message will be reset.
   // 
   // If at any point during the OFF-DELAY count down, the actual_Value returns above the reset
   // threshold (calcHystAbs), the timer will be reset to the TIME_ALM_H_OFF_DEL value, forcing 
   // the OFF-DELAY to start again.
   // ▄▄▄▄▄▄▄▄▄▄▄▄▄▄▄▄▄▄▄▄▄▄▄▄▄▄▄▄▄▄▄▄▄▄▄▄▄▄▄▄▄▄▄▄
   RUNG wire#powerrail
      Contact( #wrkAlmHEn )
      Contact( #DYNAMIC_DATA.msg_Alm_H )
      wire#w1
      { S7_Templates := "SrcType := Real" } LT_Contact(in1 := #DYNAMIC_DATA.actual_Value, in2 := #calcHystAbs)
      wire#w2
      Contact( #SYS_SIGNALS._200ms )
      Sub(in1 := #DYNAMIC_DATA.actual_Alm_H_Timer, in2 := 0.2, out => #DYNAMIC_DATA.actual_Alm_H_Timer)
   END_RUNG
   RUNG wire#w2
      { S7_Templates := "SrcType := Real" } LE_Contact(in1 := #DYNAMIC_DATA.actual_Alm_H_Timer, in2 := 0.0)
      R_Coil( #DYNAMIC_DATA.msg_Alm_H )
   END_RUNG
   RUNG wire#w1
      { S7_Templates := "SrcType := Real" } GE_Contact(in1 := #DYNAMIC_DATA.actual_Value, in2 := #calcHystAbs)
      { S7_GenerateENO := "TRUE" } Move(in := #STATIC_DATA.TIME_ALM_H_OFF_DEL, out1 => #DYNAMIC_DATA.actual_Alm_H_Timer)
   END_RUNG
   // the same network as SCL:
   #_w1 := #wrkAlmHEn AND #DYNAMIC_DATA.msg_Alm_H;
   #_w2 := #_w1 AND (#DYNAMIC_DATA.actual_Value < #calcHystAbs);
   IF #_w2 AND #SYS_SIGNALS._200ms THEN
       #DYNAMIC_DATA.actual_Alm_H_Timer := #DYNAMIC_DATA.actual_Alm_H_Timer - 0.2;
   END_IF;
   IF #_w2 AND (#DYNAMIC_DATA.actual_Alm_H_Timer <= 0.0) THEN #DYNAMIC_DATA.msg_Alm_H := FALSE; END_IF;
   IF #_w1 AND (#DYNAMIC_DATA.actual_Value >= #calcHystAbs) THEN
       #DYNAMIC_DATA.actual_Alm_H_Timer := #STATIC_DATA.TIME_ALM_H_OFF_DEL;
   END_IF;
END_REGION

REGION Network 25: Low alarm — Ensure hysteresis is not negative (error check)
   // ▀▀▀▀▀▀▀▀▀▀▀▀▀▀▀▀▀▀▀▀▀▀▀▀▀▀▀▀▀▀▀▀▀▀▀▀▀▀▀▀▀▀▀▀
   // The hysteresis value must not be a negative number. If it is, it is a value of zero is used in
   // its place.
   // 
   // wrkHyst holds the value of the hysteresis signal being applied, this will either be 
   // SP_ALM_L_HYST_VAL or zero (if SP_ALM_L_HYST_VAL were set to a negative value)
   // 
   // calcHystAbs holds the absolute value of the alarm reset threshold, for low alarms this is:
   // ┌─────────────────────┐
   // │ calcHystAbs = SP_ALM_L_VAL ┼ wrkHyst     │
   // └─────────────────────┘
   // 
   // The two threshold values for the low alarm are thus:
   // 
   //      Low alarm activation threshold = SP_ALM_L_VAL
   //      Low alarm reset threshold          = calcHystAbs
   // 
   // Note:    The hysteresis is only checked if alarm is being evaluated
   // ▄▄▄▄▄▄▄▄▄▄▄▄▄▄▄▄▄▄▄▄▄▄▄▄▄▄▄▄▄▄▄▄▄▄▄▄▄▄▄▄▄▄▄▄
   RUNG wire#powerrail
      Contact( #wrkAlmLEn )
      wire#w1
      { S7_GenerateENO := "TRUE" } Move(in := #STATIC_DATA.SP_ALM_L_HYST_VAL, out1 => #wrkHyst)
   END_RUNG
   RUNG wire#w1
      { S7_Templates := "SrcType := Real" } LT_Contact(in1 := #STATIC_DATA.SP_ALM_L_HYST_VAL, in2 := 0.0)
      { S7_GenerateENO := "TRUE" } Move(in := 0.0, out1 => #wrkHyst)
   END_RUNG
   RUNG wire#w1
      Add(in1 := #STATIC_DATA.SP_ALM_L_VAL, in2 := #wrkHyst, out => #calcHystAbs)
   END_RUNG
   // the same network as SCL:
   IF #wrkAlmLEn THEN #wrkHyst := #STATIC_DATA.SP_ALM_L_HYST_VAL; END_IF;
   IF #wrkAlmLEn AND (#STATIC_DATA.SP_ALM_L_HYST_VAL < 0.0) THEN #wrkHyst := 0.0; END_IF;
   IF #wrkAlmLEn THEN #calcHystAbs := #STATIC_DATA.SP_ALM_L_VAL + #wrkHyst; END_IF;
END_REGION

REGION Network 26: Low alarm — Check for activation level and ON-DELAY timer
   // ▀▀▀▀▀▀▀▀▀▀▀▀▀▀▀▀▀▀▀▀▀▀▀▀▀▀▀▀▀▀▀▀▀▀▀▀▀▀▀▀▀▀▀▀
   // If the low alarm has been enabled and is not masked and the actual_Value is less than or 
   // equal to the alarm setpoint (SP_ALM_L_VAL), but the alarm has not yet been triggered 
   // (msg_Alm_L = 0) then the ON-DELAY phase is active (the alarm timer is counting down).
   // 
   // The timer will begin to count down from the value in TIME_ALM_L_ON_DEL using the 200ms 
   // pulse (it will count down in increments of 0.2s). If the Low alarm timer is less than or equal to 
   // zero, then the ON-DELAY has expired and the Low Alarm message will become active.
   // 
   // If at any point during the ON-DELAY count down, the actual_Value rises above the activation
   // setpoint (SP_ALM_L_VAL), the timer will be reset to the TIME_ALM_L_ON_DEL value, forcing 
   // the ON-DELAY to start again.
   // ▄▄▄▄▄▄▄▄▄▄▄▄▄▄▄▄▄▄▄▄▄▄▄▄▄▄▄▄▄▄▄▄▄▄▄▄▄▄▄▄▄▄▄▄
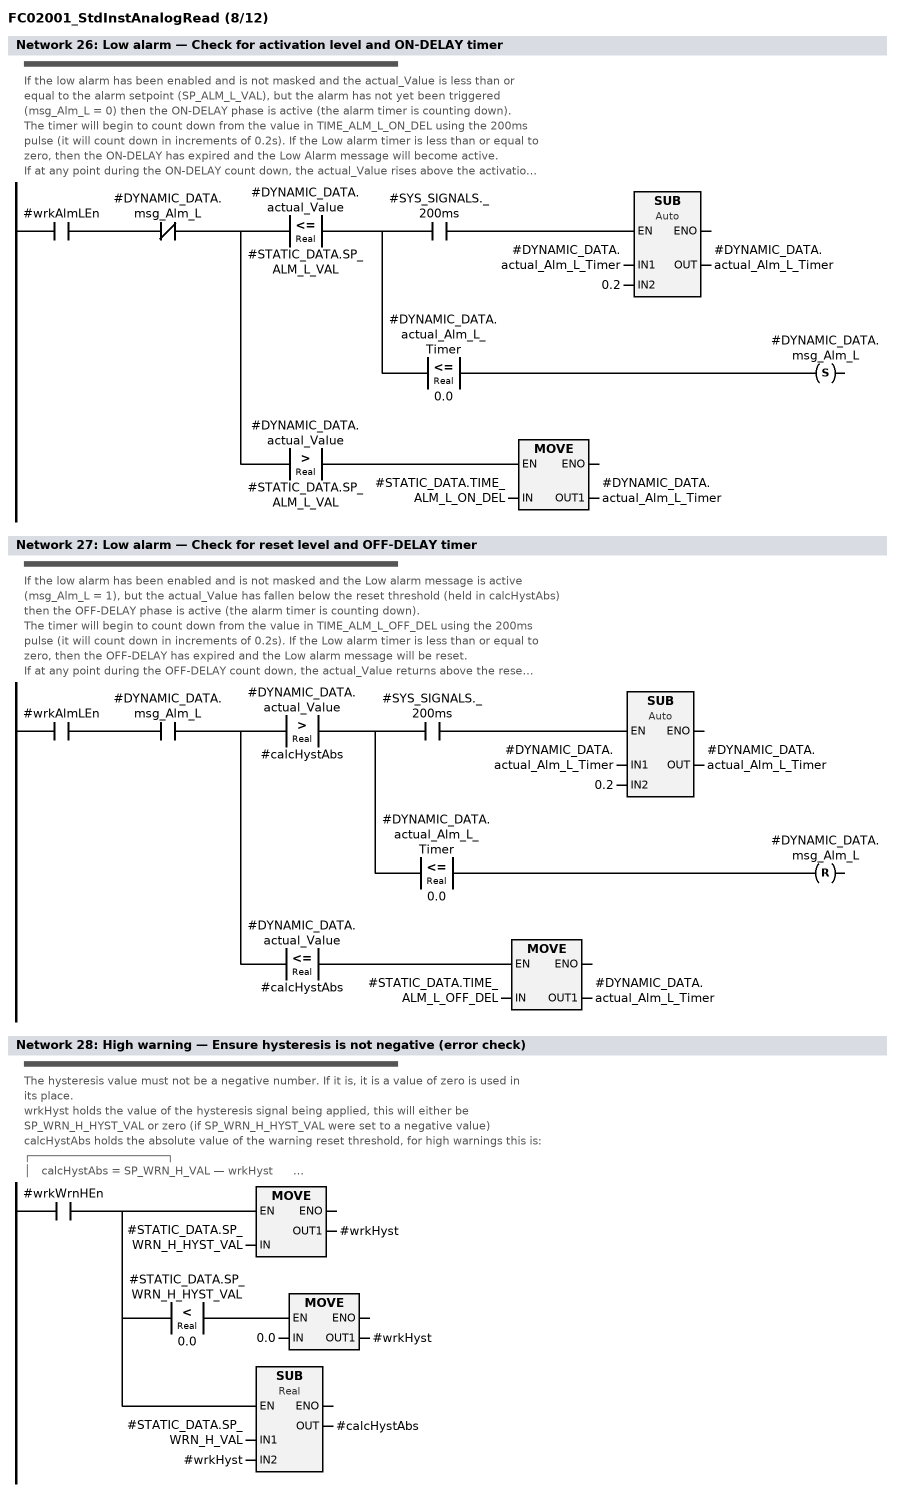
   RUNG wire#powerrail
      Contact( #wrkAlmLEn )
      I_Contact( #DYNAMIC_DATA.msg_Alm_L )
      wire#w1
      { S7_Templates := "SrcType := Real" } LE_Contact(in1 := #DYNAMIC_DATA.actual_Value, in2 := #STATIC_DATA.SP_ALM_L_VAL)
      wire#w2
      Contact( #SYS_SIGNALS._200ms )
      Sub(in1 := #DYNAMIC_DATA.actual_Alm_L_Timer, in2 := 0.2, out => #DYNAMIC_DATA.actual_Alm_L_Timer)
   END_RUNG
   RUNG wire#w2
      { S7_Templates := "SrcType := Real" } LE_Contact(in1 := #DYNAMIC_DATA.actual_Alm_L_Timer, in2 := 0.0)
      S_Coil( #DYNAMIC_DATA.msg_Alm_L )
   END_RUNG
   RUNG wire#w1
      { S7_Templates := "SrcType := Real" } GT_Contact(in1 := #DYNAMIC_DATA.actual_Value, in2 := #STATIC_DATA.SP_ALM_L_VAL)
      { S7_GenerateENO := "TRUE" } Move(in := #STATIC_DATA.TIME_ALM_L_ON_DEL, out1 => #DYNAMIC_DATA.actual_Alm_L_Timer)
   END_RUNG
   // the same network as SCL:
   #_w1 := #wrkAlmLEn AND NOT #DYNAMIC_DATA.msg_Alm_L;
   #_w2 := #_w1 AND (#DYNAMIC_DATA.actual_Value <= #STATIC_DATA.SP_ALM_L_VAL);
   IF #_w2 AND #SYS_SIGNALS._200ms THEN
       #DYNAMIC_DATA.actual_Alm_L_Timer := #DYNAMIC_DATA.actual_Alm_L_Timer - 0.2;
   END_IF;
   IF #_w2 AND (#DYNAMIC_DATA.actual_Alm_L_Timer <= 0.0) THEN #DYNAMIC_DATA.msg_Alm_L := TRUE; END_IF;
   IF #_w1 AND (#DYNAMIC_DATA.actual_Value > #STATIC_DATA.SP_ALM_L_VAL) THEN
       #DYNAMIC_DATA.actual_Alm_L_Timer := #STATIC_DATA.TIME_ALM_L_ON_DEL;
   END_IF;
END_REGION

REGION Network 27: Low alarm — Check for reset level and OFF-DELAY timer
   // ▀▀▀▀▀▀▀▀▀▀▀▀▀▀▀▀▀▀▀▀▀▀▀▀▀▀▀▀▀▀▀▀▀▀▀▀▀▀▀▀▀▀▀▀
   // If the low alarm has been enabled and is not masked and the Low alarm message is active 
   // (msg_Alm_L = 1), but the actual_Value has fallen below the reset threshold (held in calcHystAbs) 
   // then the OFF-DELAY phase is active (the alarm timer is counting down).
   // 
   // The timer will begin to count down from the value in TIME_ALM_L_OFF_DEL using the 200ms 
   // pulse (it will count down in increments of 0.2s). If the Low alarm timer is less than or equal to 
   // zero, then the OFF-DELAY has expired and the Low alarm message will be reset.
   // 
   // If at any point during the OFF-DELAY count down, the actual_Value returns above the reset
   // threshold (calcHystAbs), the timer will be reset to the TIME_ALM_L_OFF_DEL value, forcing 
   // the OFF-DELAY to start again.
   // ▄▄▄▄▄▄▄▄▄▄▄▄▄▄▄▄▄▄▄▄▄▄▄▄▄▄▄▄▄▄▄▄▄▄▄▄▄▄▄▄▄▄▄▄
   RUNG wire#powerrail
      Contact( #wrkAlmLEn )
      Contact( #DYNAMIC_DATA.msg_Alm_L )
      wire#w1
      { S7_Templates := "SrcType := Real" } GT_Contact(in1 := #DYNAMIC_DATA.actual_Value, in2 := #calcHystAbs)
      wire#w2
      Contact( #SYS_SIGNALS._200ms )
      Sub(in1 := #DYNAMIC_DATA.actual_Alm_L_Timer, in2 := 0.2, out => #DYNAMIC_DATA.actual_Alm_L_Timer)
   END_RUNG
   RUNG wire#w2
      { S7_Templates := "SrcType := Real" } LE_Contact(in1 := #DYNAMIC_DATA.actual_Alm_L_Timer, in2 := 0.0)
      R_Coil( #DYNAMIC_DATA.msg_Alm_L )
   END_RUNG
   RUNG wire#w1
      { S7_Templates := "SrcType := Real" } LE_Contact(in1 := #DYNAMIC_DATA.actual_Value, in2 := #calcHystAbs)
      { S7_GenerateENO := "TRUE" } Move(in := #STATIC_DATA.TIME_ALM_L_OFF_DEL, out1 => #DYNAMIC_DATA.actual_Alm_L_Timer)
   END_RUNG
   // the same network as SCL:
   #_w1 := #wrkAlmLEn AND #DYNAMIC_DATA.msg_Alm_L;
   #_w2 := #_w1 AND (#DYNAMIC_DATA.actual_Value > #calcHystAbs);
   IF #_w2 AND #SYS_SIGNALS._200ms THEN
       #DYNAMIC_DATA.actual_Alm_L_Timer := #DYNAMIC_DATA.actual_Alm_L_Timer - 0.2;
   END_IF;
   IF #_w2 AND (#DYNAMIC_DATA.actual_Alm_L_Timer <= 0.0) THEN #DYNAMIC_DATA.msg_Alm_L := FALSE; END_IF;
   IF #_w1 AND (#DYNAMIC_DATA.actual_Value <= #calcHystAbs) THEN
       #DYNAMIC_DATA.actual_Alm_L_Timer := #STATIC_DATA.TIME_ALM_L_OFF_DEL;
   END_IF;
END_REGION

REGION Network 28: High warning — Ensure hysteresis is not negative (error check)
   // ▀▀▀▀▀▀▀▀▀▀▀▀▀▀▀▀▀▀▀▀▀▀▀▀▀▀▀▀▀▀▀▀▀▀▀▀▀▀▀▀▀▀▀▀
   // The hysteresis value must not be a negative number. If it is, it is a value of zero is used in
   // its place.
   // 
   // wrkHyst holds the value of the hysteresis signal being applied, this will either be 
   // SP_WRN_H_HYST_VAL or zero (if SP_WRN_H_HYST_VAL were set to a negative value)
   // 
   // calcHystAbs holds the absolute value of the warning reset threshold, for high warnings this is:
   // ┌─────────────────────┐
   // │ calcHystAbs = SP_WRN_H_VAL — wrkHyst    │
   // └─────────────────────┘
   // 
   // The two threshold values for the high warning are thus:
   // 
   //      High warning activation threshold = SP_WRN_H_VAL
   //      High warning reset threshold          = calcHystAbs
   // 
   // Note:    The hysteresis is only checked if warning is being evaluated
   // ▄▄▄▄▄▄▄▄▄▄▄▄▄▄▄▄▄▄▄▄▄▄▄▄▄▄▄▄▄▄▄▄▄▄▄▄▄▄▄▄▄▄▄▄
   RUNG wire#powerrail
      Contact( #wrkWrnHEn )
      wire#w1
      { S7_GenerateENO := "TRUE" } Move(in := #STATIC_DATA.SP_WRN_H_HYST_VAL, out1 => #wrkHyst)
   END_RUNG
   RUNG wire#w1
      { S7_Templates := "SrcType := Real" } LT_Contact(in1 := #STATIC_DATA.SP_WRN_H_HYST_VAL, in2 := 0.0)
      { S7_GenerateENO := "TRUE" } Move(in := 0.0, out1 => #wrkHyst)
   END_RUNG
   RUNG wire#w1
      { S7_Templates := "SrcType := Real"; S7_GenerateENO := "TRUE" } Sub(in1 := #STATIC_DATA.SP_WRN_H_VAL, in2 := #wrkHyst, out => #calcHystAbs)
   END_RUNG
   // the same network as SCL:
   IF #wrkWrnHEn THEN #wrkHyst := #STATIC_DATA.SP_WRN_H_HYST_VAL; END_IF;
   IF #wrkWrnHEn AND (#STATIC_DATA.SP_WRN_H_HYST_VAL < 0.0) THEN #wrkHyst := 0.0; END_IF;
   IF #wrkWrnHEn THEN #calcHystAbs := #STATIC_DATA.SP_WRN_H_VAL - #wrkHyst; END_IF;
END_REGION

